	        ELSIF
	            #sx_PreStartManual                                                          // IF in manual jog mode
	            AND (NOT #iq_UDT_EquipmentControl.Request.SignalingRequest                  // Signaling request done
	            OR #Jog_Enable.qx_DelayedSignal)
	            AND NOT #sx_CombinedJogUp                                                   // If selected jog in positive direction
	            AND #sx_CombinedJogDown                                                     // and there is command to jog in negative direction
	        THEN

	            #sx_JogUp := FALSE;                                                         // reset jog positive
	            #sx_JogDown := TRUE;                                                        // set jog negative
	            #sx_Jog := true;

	        ELSIF
	            NOT #sx_PreStartManual                                                      // If not in manual mode
	            OR (#sx_PreStartManual                                                      // or in manual mode
	            AND (#sx_CombinedJogUp                                                      // and jog positive is off
	            AND #sx_CombinedJogDown)                                                    // AND jog negative is off
	            OR (NOT #sx_CombinedJogUp                                                   // or jog positive is on
	            AND NOT #sx_CombinedJogDown))                                               // and jog negative is on
	        THEN

	            #sx_JogUp := FALSE;                                                         // reset jog positive
	            #sx_JogDown := FALSE;                                                       // reset jog negative
	            #sx_Jog := False;
	        END_IF;

	    END_REGION

	END_REGION

	REGION 7 - Semi automatic

	    REGION 7.1 - Semi automatic

	        IF #sx_SemiAutomatic                                                            // Not running Semi-Automatic
	            AND (#ix_ChangeModeSignal
	            AND #ii_Mode = #ci_InfeedMode)
	            AND #sx_SwitchEnable
	            AND NOT #ix_ChuteUpSensor
	        THEN

	            #sx_PreStartSemiAutomaticUp := TRUE;

	            #sx_DownRequest := FALSE;                                                   // Reset down command
	            #sx_UpRequest := TRUE;                                                      // Set up command

	        END_IF;

	        IF #sx_SemiAutomatic                                                            // Not running Semi-Automatic
	            AND (#ix_ChangeModeSignal
	            AND #ii_Mode = #ci_OutfeedMode)
	            AND #sx_SwitchEnable
	            AND NOT #ix_ChuteDownSensor
	        THEN

	            #sx_PreStartSemiAutomaticDown := TRUE;

	            #sx_DownRequest := TRUE;                                                    // Reset down command
	            #sx_UpRequest := FALSE;                                                     // Set up command

	        END_IF;

	        #R_TRIG_PreStartSemiAutomaticUp(CLK := #sx_PreStartSemiAutomaticUp);
	        #R_TRIG_PreStartSemiAutomaticDown(CLK := #sx_PreStartSemiAutomaticDown);

	        //Set Signaling Request
	        IF #R_TRIG_PreStartSemiAutomaticUp.Q OR #R_TRIG_PreStartSemiAutomaticDown.Q THEN
	            #iq_UDT_EquipmentControl.Request.SignalingRequest := TRUE;
	        END_IF;

	        IF #sx_SemiAutomatic
	            AND (#ix_ChuteUpSensor
	            AND #sx_UpRequest)
	            OR #s_UDT_HMIStatus.Specific.SwitchingTimerError
	        THEN
	            #sx_UpRequest := false;
	            #sx_PreStartSemiAutomaticUp := false;
	        END_IF;

	        IF #sx_SemiAutomatic
	            AND (NOT #ix_LiftDownSensor
	            AND #sx_DownRequest)
	            OR #s_UDT_HMIStatus.Specific.SwitchingTimerError
	        THEN
	            #sx_DownRequest := false;
	            #sx_PreStartSemiAutomaticDown := false;
	        END_IF;

	    END_REGION

	    REGION 7.2 - Stop conveyor

	        #qx_ExternalHold := #ss_ColumLiftInterface.Positioning;                                            // External stop signal

	    END_REGION

	END_REGION

	REGION 8 - Write interface DB signals

	    REGION 8.1 - Signal interface

	        #iq_UDT_LiftInterface.InternalErrorReset := #iq_UDT_EquipmentControl.Command.Reset;      // Write Reset signal to the VFD interface
	        #iq_UDT_LiftInterface.ResetStatistics := #iq_UDT_EquipmentControl.Command.ResetData;     // Write Reset data signal to the VFD interface

	    END_REGION

	    REGION 8.1 - Mode selection

	        #ss_ColumLiftInterface.SemiAutomatic :=
	        (#sx_SemiAutomatic                                                               // Automatic started
	        OR #sx_Stopping);                                                                // stopping is activated Go to default position

	        #ss_ColumLiftInterface.Manual :=                                                         // Manual mode is started
	        #sx_CombinedJogUp                                                           // IF selected jog in positive direction
	        OR #sx_CombinedJogDown;

	    END_REGION

	    REGION 8.2 - Run enable

	        #ss_ColumLiftInterface.RunEnabled :=                                                  // Enable the positioning device to run
	        NOT #iq_UDT_LiftInterface.InternalErrorVFD                               // or there are errors in the VFD
	        AND NOT #sx_ConfigurationError                                                   // configuration is wrong
	        AND #ix_HardwareOk                                                        // or an internal error in the RIO panel occured
	        AND (#ss_ColumLiftInterface.SemiAutomatic                                             // VSU is in semi-automatic mode
	        OR (#ss_ColumLiftInterface.Manual                                                     // manual mode is active
	        AND (#sx_CombinedJogUp                                                           // If selected jog in positive direction
	        OR #sx_CombinedJogDown)))                                                        // If selected jog in negative direction
	        AND NOT #ix_RIONotOnline;                                                       // If we don't have signal from sensors

	    END_REGION

	END_REGION

	REGION 9 - Positions reached

	    // triggers of PEC's down/up
	    #F_TRIG_PECUp(CLK := #ix_ChuteUpSensor);
	    #R_TRIG_PECUp(CLK := #ix_ChuteUpSensor);

	    #F_TRIG_PECDown(CLK := #ix_LiftDownSensor);
	    #R_TRIG_PECDown(CLK := #ix_LiftDownSensor);

	    IF #R_TRIG_PECUp.Q THEN
	        #sx_UpperPositionReached := true;
	    ELSIF (#sx_DownRequest OR #sx_JogDown) AND #F_TRIG_PECUp.Q THEN
	        #sx_UpperPositionReached := false;
	    END_IF;

	    IF #R_TRIG_PECDown.Q THEN
	        #sx_LowerPositionReached := true;
	    ELSIF (#sx_UpRequest OR #sx_JogUp) AND #F_TRIG_PECDown.Q THEN
	        #sx_LowerPositionReached := false;
	    END_IF;

	END_REGION

	REGION 10 - Run up/down

	    // Conditions to run column lift upwards
	    #iq_UDT_LiftInterface.RunRvs := ((#sx_UpRequest AND #sx_SemiAutomatic AND NOT #iq_UDT_EquipmentControl.Request.SignalingRequest)
	    OR #sx_JogUp)
	    AND (NOT #sx_UpperPositionReached OR (#sx_MaintenanceControl AND #sx_JogUp))
	    AND #ss_ColumLiftInterface.RunEnabled
	    AND #ix_LiftUpSensor;

	    // Conditions to run column lift down
	    #iq_UDT_LiftInterface.RunFwd := ((#sx_DownRequest AND #sx_SemiAutomatic AND NOT #iq_UDT_EquipmentControl.Request.SignalingRequest)
	    OR #sx_JogDown)
	    AND #ss_ColumLiftInterface.RunEnabled
	    AND #ix_LiftDownSensor;

	END_REGION

	REGION 11 - Column lift speed

	    IF #ss_ColumLiftInterface.Manual THEN
	        #iq_UDT_LiftInterface.SpeedSetpoint := #i_UDT_ColumnLiftConfiguration.ManualModeSpeed;
	    ELSE
	        #iq_UDT_LiftInterface.SpeedSetpoint := #i_UDT_ColumnLiftConfiguration.NominalSpeedSetPoint;
	    END_IF;

	END_REGION

	REGION 12 - Statistics

	    // Down Time
	    IF #sx_SemiAutomatic                                                                 // Automatic active
	        AND NOT #sx_Ready                                                                // Conveyor not ready
	        OR #iq_UDT_EquipmentControl.Command.ResetData                                    // Reset statistics
	    THEN

	        "FC_Statistics"(ix_Reset := #iq_UDT_EquipmentControl.Command.ResetData,              // Or reset statistics from control
	                        ix_Activate := #sx_SemiAutomatic AND NOT #sx_Ready,                  // VSU is stopped
	                        ix_RTrigActivate := #R_TRIG_DownTime.Q,                              // VSU is stopped triger
	                        iqUDT_Statistics := #iq_UDT_Statistics.DownTime);                   // VSU is stopped statistics
	    END_IF;

	    // Up time
	    IF #sx_SemiAutomatic                                // Automatic active
	        AND #sx_Ready                                   // Ready active
	        OR #iq_UDT_EquipmentControl.Command.ResetData   // Reset statistics
	    THEN
	        "FC_Statistics"(ix_Reset := #iq_UDT_EquipmentControl.Command.ResetData,        // OR reset statistics from control
	                        ix_Activate := #sx_SemiAutomatic AND #sx_Ready,                // VSU is running
	                        ix_RTrigActivate := #R_TRIG_UpTime.Q,                          // VSU running trigger
	                        iqUDT_Statistics := #iq_UDT_Statistics.UpTime);               // VSU running statistics

	    END_IF;

	END_REGION

	REGION 13 - Status

	    #s_UDT_Status.Stopped := #sx_Ready AND NOT #sx_SemiAutomatic AND NOT #sx_Stopping;      // stopped
	    #s_UDT_Status.AutoON := #sx_SemiAutomatic OR #sx_Stopping;                              // Auto On
	    #s_UDT_Status.Halted := FALSE;                                                          // Halted
	    #s_UDT_Status.Dieback := FALSE;                                                         // Die back
	    #s_UDT_Status.Running := (#sx_UpRequest OR #sx_DownRequest) AND #sx_SemiAutomatic;      // Running
	    #s_UDT_Status.ManualRun := #ix_SS_Man AND #iq_UDT_LiftInterface.VFDRunning;            // Manual run
	    #s_UDT_Status.Manual := #ix_SS_Man;                                                     // Manual
	    #s_UDT_Status.EnergySave := FALSE;                                                      // Energy save active
	    #s_UDT_Status.SafetyStop := NOT #ix_SafetyOk;                                           // Safety not ok

	    //   Specific status
	    IF #s_UDT_StatusOld <> #s_UDT_Status                                            // update on change
	    THEN

	        // Set status to status number
	        #s_UDT_HMIStatus.Status := 0;                                               // Initialise status number

	        IF #s_UDT_Status.Running                                                    // Running in semi automatic
	        THEN

	            #s_UDT_HMIStatus.Status := "DB_HMIStatusConfiguration".PositionChangeOngoing;

	        END_IF;

	        IF #s_UDT_Status.Stopped                                                    // Stopped
	        THEN

	            #s_UDT_HMIStatus.Status := "DB_HMIStatusConfiguration".Stopped;

	        END_IF;

	        IF #s_UDT_Status.AutoON                                                   // Dieback
	        THEN

	            #s_UDT_HMIStatus.Status := "DB_HMIStatusConfiguration".AutoON;

	        END_IF;

	        IF #s_UDT_Status.ManualRun                                                  // Manual run
	        THEN

	            #s_UDT_HMIStatus.Status := "DB_HMIStatusConfiguration".ManualRun;

	        END_IF;

	        IF #s_UDT_Status.Manual                                                     // Manual
	        THEN

	            #s_UDT_HMIStatus.Status := "DB_HMIStatusConfiguration".Manual;

	        END_IF;

	        IF #iq_UDT_LiftInterface.InternalWarningVFD                                  // The VFD has an internal warning

	        THEN

	            #s_UDT_HMIStatus.Status := "DB_HMIStatusConfiguration".Warning;

	        END_IF;

	        IF #s_UDT_Status.Error                                 // The VFD has an internal warning
	        THEN
	            #s_UDT_HMIStatus.Status := "DB_HMIStatusConfiguration".Error;
	        END_IF;

	        IF #s_UDT_Status.SafetyStop                                                 // Safety stop
	        THEN

	            #s_UDT_HMIStatus.Status := "DB_HMIStatusConfiguration".SafetyStop;

	        END_IF;


	        #s_UDT_StatusOld := #s_UDT_Status;                                          // Copy status TO memory
	        #q_UDT_Status := #s_UDT_Status;                                             // Copy status to output

	    END_IF;

	    //Actual position
	    #s_UDT_HMIStatus.Specific.UpperPosition := #ix_ChuteUpSensor;
	    #s_UDT_HMIStatus.Specific.LowerPosition := NOT #ix_LiftDownSensor;                  //Lower position was changed to use limit switch down because of the project specyfic equipment

	    //Limit switch active
	    IF #sx_LiftUpFiltered AND NOT #ix_RIONotOnline THEN

	        #s_UDT_HMIStatus.Specific.LimitSensorUpperPosition := True;

	    END_IF;

	(*    IF NOT #ix_LiftDownSensor THEN

	        #s_UDT_HMIStatus.Specific.LimitSensorLowerPosition := True;

	    END_IF; *)

	    IF #sx_MaintenanceControl THEN

	        #s_UDT_HMIStatus.Specific.MaintenaceModeActive := True;

	    END_IF;

	    #q_UDT_HMIStatus := #s_UDT_HMIStatus;                                       // Copy status to output

	END_REGION

	REGION 14 - Report to control block

	    #iq_UDT_EquipmentControl.Request.InhibitStop := #iq_UDT_EquipmentControl.Request.InhibitStop OR #ss_ColumLiftInterface.Positioning;

	    "FC_EquipmentReport"(iUDT_Status := #s_UDT_Status,
	                         iqUDT_Control := #iq_UDT_EquipmentControl);

	END_REGION

	REGION 15 - Internal errors and warnings reset

	    #iq_UDT_LiftInterface.InternalErrorPEC := FALSE;
	    #iq_UDT_LiftInterface.InternalWarningTracking := FALSE;
	    #iq_UDT_LiftInterface.InternalErrorTracking := FALSE;
	    #iq_UDT_LiftInterface.InternalWarningVFD := FALSE;
	    #iq_UDT_LiftInterface.InternalErrorVFD := FALSE;
	    #iq_UDT_LiftInterface.Disconnected := FALSE;

	END_REGION

END_FUNCTION_BLOCK

FUNCTION_BLOCK "FB_CodingBeltModes"
{ S7_Optimized_Access := 'TRUE' }
VERSION : 0.1
// ATTRIBUTES
// AUTO_NUMBER = True
// BLOCK_NUMBER = 90
// END_ATTRIBUTES
   VAR_INPUT
      i_UDT_Configuration { ExternalAccessible := 'False'; ExternalVisible := 'False'; ExternalWritable := 'False'} : "UDT_CodingBeltModesConfiguration";   // Function configuration
      ii_Displacement { ExternalAccessible := 'False'; ExternalVisible := 'False'; ExternalWritable := 'False'} : Int;   // Conveyor displacement in one PLC cycle [cm]
      ix_KneeButton { ExternalAccessible := 'False'; ExternalVisible := 'False'; ExternalWritable := 'False'} : Bool;   // Knee button
      ix_LabellingMode { ExternalAccessible := 'False'; ExternalVisible := 'False'; ExternalWritable := 'False'} : Bool;   // Local switch Labeling mode
      ix_ContinueMode { ExternalAccessible := 'False'; ExternalVisible := 'False'; ExternalWritable := 'False'} : Bool;   // Local switch Continue mode
      ix_BufferMode { ExternalAccessible := 'False'; ExternalVisible := 'False'; ExternalWritable := 'False'} : Bool;   // Local switch Buffer mode
      ix_LineModeInfeed { ExternalAccessible := 'False'; ExternalVisible := 'False'; ExternalWritable := 'False'} : Bool;   // Interface with main line - bool or new UDT??? Infeed and Outfeed?
      ix_LineModeOutfeed { ExternalAccessible := 'False'; ExternalVisible := 'False'; ExternalWritable := 'False'} : Bool;   // Interface with main line - bool or new UDT??? Infeed and Outfeed?
      ix_PEC_BoS { ExternalAccessible := 'False'; ExternalVisible := 'False'; ExternalWritable := 'False'} : Bool;   // BoS sensor
      ix_PEC_EoS { ExternalAccessible := 'False'; ExternalVisible := 'False'; ExternalWritable := 'False'} : Bool;   // EoS sensor
   END_VAR

   VAR_OUTPUT
      q_UDT_HMIStatus { ExternalAccessible := 'False'; ExternalVisible := 'False'; ExternalWritable := 'False'} : "UDT_CodingBeltModesStatus";   // Status
      qx_RequestHold_Conveyor { ExternalAccessible := 'False'; ExternalVisible := 'False'; ExternalWritable := 'False'} : Bool;   // Request hold for conveyor
   END_VAR

   VAR
      R_TRIG_KneeButton {InstructionName := 'R_TRIG'; LibVersion := '1.0'; ExternalAccessible := 'False'; ExternalVisible := 'False'; ExternalWritable := 'False'; S7_SetPoint := 'False'} : R_TRIG;   // Rising edge trigger of toogle button
      R_TRIG_LabellingMode {InstructionName := 'R_TRIG'; LibVersion := '1.0'; ExternalAccessible := 'False'; ExternalVisible := 'False'; ExternalWritable := 'False'; S7_SetPoint := 'False'} : R_TRIG;   // Rising edge trigger of labelling mode
      R_TRIG_ContinueMode {InstructionName := 'R_TRIG'; LibVersion := '1.0'; ExternalAccessible := 'False'; ExternalVisible := 'False'; ExternalWritable := 'False'; S7_SetPoint := 'False'} : R_TRIG;   // Rising edge trigger of continue mode
      R_TRIG_BufferMode {InstructionName := 'R_TRIG'; LibVersion := '1.0'; ExternalAccessible := 'False'; ExternalVisible := 'False'; ExternalWritable := 'False'; S7_SetPoint := 'False'} : R_TRIG;   // Rising edge trigger of buffer mode
      R_TRIG_LineModeInfeed {InstructionName := 'R_TRIG'; LibVersion := '1.0'; ExternalAccessible := 'False'; ExternalVisible := 'False'; ExternalWritable := 'False'; S7_SetPoint := 'False'} : R_TRIG;   // Rising edge trigger of Infeed mode
      R_TRIG_LineModeOutfeed {InstructionName := 'R_TRIG'; LibVersion := '1.0'; ExternalAccessible := 'False'; ExternalVisible := 'False'; ExternalWritable := 'False'; S7_SetPoint := 'False'} : R_TRIG;   // Rising edge trigger of Outfeed mode
      F_TRIG_PEC_BoS {InstructionName := 'F_TRIG'; LibVersion := '1.0'; ExternalAccessible := 'False'; ExternalVisible := 'False'; ExternalWritable := 'False'; S7_SetPoint := 'False'} : F_TRIG;   // Falling edge trigger of sensor
      F_TRIG_PEC_EoS {InstructionName := 'F_TRIG'; LibVersion := '1.0'; ExternalAccessible := 'False'; ExternalVisible := 'False'; ExternalWritable := 'False'; S7_SetPoint := 'False'} : F_TRIG;
      sx_LabellingMode { ExternalAccessible := 'False'; ExternalVisible := 'False'; ExternalWritable := 'False'} : Bool;   // Labelling Mode
      sx_ContinueMode { ExternalAccessible := 'False'; ExternalVisible := 'False'; ExternalWritable := 'False'} : Bool;   // Continue Mode
      sx_BufferMode { ExternalAccessible := 'False'; ExternalVisible := 'False'; ExternalWritable := 'False'} : Bool;   // Buffer Mode
      sx_RequestHold { ExternalAccessible := 'False'; ExternalVisible := 'False'; ExternalWritable := 'False'} : Bool;   // Request hold for conveyor
      sx_GeneralError { ExternalAccessible := 'False'; ExternalVisible := 'False'; ExternalWritable := 'False'} : Bool;   // General error
      sx_ConfigurationError { ExternalAccessible := 'False'; ExternalVisible := 'False'; ExternalWritable := 'False'} : Bool;   // Configuration error
      sx_CountDistance { ExternalAccessible := 'False'; ExternalVisible := 'False'; ExternalWritable := 'False'} : Bool;   // Start counting distance to stop position
      sx_ParcelAtPosition { ExternalAccessible := 'False'; ExternalVisible := 'False'; ExternalWritable := 'False'} : Bool;   // The parcel has reached the position
      si_DistanceToStopPosition { ExternalAccessible := 'False'; ExternalVisible := 'False'; ExternalWritable := 'False'} : Int;   // Distance to stop position
   END_VAR


BEGIN
	(*
	----------------------------------------------------------------------------------------
	|                                                                                      |
	|  Copyright  2023             Fortna Europe BV                                        |
	|  All Rights Reserved         Netherlands                                             |
	|                                                                                      |
	|                                                                                      |
	----------------------------------------------------------------------------------------

	Version history:
	Date        | Version   | Author       | Remark
	----------------------------------------------------------------------------------------
	27/07/2023  | 1.0       | S. Nikodem   | Release TIA 17  | DHL Munich 2023
	06/10/2023  | 1.1       | M.Diebel     | Status handling | DHL Munich 2023
	04.12/2023  | 1.2       | M.Diebel     | Stop status     | DHL Munich 2023
	12/03/2024  | 1.3       | S. Nieswiec  | Added to new Baseline
	*)

	REGION 1 - Triggers

	    //Knee button
	    #R_TRIG_KneeButton(CLK := (#ix_KneeButton));

	    //Detect end of the parcel
	    //BoS
	    #F_TRIG_PEC_BoS(CLK := #ix_PEC_BoS);
	    //EoS
	    #F_TRIG_PEC_EoS(CLK := #ix_PEC_EoS);

	END_REGION

	REGION 2 - Error detection

	    // Only one mode can be active
	    IF (#ix_LabellingMode AND #ix_ContinueMode)
	        OR (#ix_LabellingMode AND #ix_BufferMode)
	        OR (#ix_ContinueMode AND #ix_BufferMode)
	    THEN

	        #sx_GeneralError := TRUE;

	    ELSE

	        #sx_GeneralError := False;

	    END_IF;

	    //Configuration Error
	    IF #i_UDT_Configuration.LabellingMode_ParcelStop <= 0 THEN

	        #sx_ConfigurationError := TRUE;

	    ELSE

	        #sx_ConfigurationError := False;

	    END_IF;

	END_REGION

	REGION 3 - Modes

	    // Select mode - when the local switch is used or the main line mode is changed

	    #R_TRIG_LabellingMode(CLK := #ix_LabellingMode AND NOT #sx_BufferMode);

	    #R_TRIG_ContinueMode(CLK := #ix_ContinueMode);

	    #R_TRIG_BufferMode(CLK := #ix_BufferMode AND NOT #sx_LabellingMode);

	    #R_TRIG_LineModeInfeed(CLK := #ix_LineModeInfeed);

	    #R_TRIG_LineModeOutfeed(CLK := #ix_LineModeOutfeed);

	    IF #R_TRIG_LabellingMode.Q
	        OR #R_TRIG_ContinueMode.Q
	        OR #R_TRIG_BufferMode.Q
	        OR #R_TRIG_LineModeInfeed.Q
	        OR #R_TRIG_LineModeOutfeed.Q
	    THEN

	        //Clean value from variable when new mode is selected.
	        #sx_LabellingMode := FALSE;
	        #sx_ContinueMode := FALSE;
	        #sx_BufferMode := FALSE;

	        #sx_CountDistance := FALSE;
	        #si_DistanceToStopPosition := 0;
	        #sx_ParcelAtPosition := FALSE;
	        #sx_RequestHold := FALSE;

	        //
	        IF #ix_LabellingMode AND
	            ((#i_UDT_Configuration.Infeed.LabellingMode AND #ix_LineModeInfeed)
	            OR (#i_UDT_Configuration.Outfeed.LabellingMode AND #ix_LineModeOutfeed))
	        THEN

	            #sx_LabellingMode := True;

	        ELSIF
	            #ix_ContinueMode AND
	            ((#i_UDT_Configuration.Infeed.ContinueMode AND #ix_LineModeInfeed)
	            OR (#i_UDT_Configuration.Outfeed.ContinueMode AND #ix_LineModeOutfeed))
	        THEN

	            #sx_ContinueMode := True;

	        ELSIF
	            #ix_BufferMode AND
	            ((#i_UDT_Configuration.Infeed.BufferMode AND #ix_LineModeInfeed)
	            OR (#i_UDT_Configuration.Outfeed.BufferMode AND #ix_LineModeOutfeed))
	        THEN

	            #sx_BufferMode := True;

	        END_IF;

	    END_IF;

	    REGION 3.1 - Labelling mode

	        IF #sx_LabellingMode THEN

	            IF (#F_TRIG_PEC_BoS.Q AND #ix_LineModeInfeed) OR (#F_TRIG_PEC_EoS.Q AND #ix_LineModeOutfeed) THEN

	                #sx_CountDistance := TRUE;

	            END_IF;

	            //Count the distance to stop parcel position
	            IF #sx_CountDistance THEN

	                #si_DistanceToStopPosition += ABS(#ii_Displacement);

	                IF #si_DistanceToStopPosition > #i_UDT_Configuration.LabellingMode_ParcelStop THEN

	                    #sx_CountDistance := FALSE;
	                    #si_DistanceToStopPosition := 0;
	                    #sx_ParcelAtPosition := True;

	                END_IF;

	            END_IF;

	            //When parcel is at position then stop conveyor
	            #sx_RequestHold := #sx_ParcelAtPosition;

	            //Operator confirm the parcel using knee button
	            IF #R_TRIG_KneeButton.Q THEN

	                #sx_ParcelAtPosition := False;

	            END_IF;


	        END_IF;

	    END_REGION

	    REGION 3.2 - Continue mode

	        IF #sx_ContinueMode THEN

	            IF #R_TRIG_KneeButton.Q THEN

	                #sx_RequestHold := NOT #sx_RequestHold;

	            END_IF;

	        END_IF;

	    END_REGION
	END_REGION

	REGION 4 - Status

	    //Selected mode
	    #q_UDT_HMIStatus.Specific.Infeed_LabellingMode := #sx_LabellingMode AND #ix_LineModeInfeed;
	    #q_UDT_HMIStatus.Specific.Infeed_ContinueMode := #sx_ContinueMode AND #ix_LineModeInfeed;
	    #q_UDT_HMIStatus.Specific.Infeed_BufferMode := #sx_BufferMode AND #ix_LineModeInfeed;
	    #q_UDT_HMIStatus.Specific.Outfeed_LabellingMode := #sx_LabellingMode AND #ix_LineModeOutfeed;
	    #q_UDT_HMIStatus.Specific.Outfeed_ContinueMode := #sx_ContinueMode AND #ix_LineModeOutfeed;
	    #q_UDT_HMIStatus.Specific.Outfeed_BufferMode := #sx_BufferMode AND #ix_LineModeOutfeed;

	    IF (#sx_LabellingMode AND #ix_LineModeInfeed) OR (#sx_LabellingMode AND #ix_LineModeOutfeed)
	    THEN

	        #q_UDT_HMIStatus.Status := "DB_HMIStatusConfiguration".LabbelingMode;

	    END_IF;

	    IF (#sx_ContinueMode AND #ix_LineModeInfeed) OR (#sx_ContinueMode AND #ix_LineModeOutfeed)
	    THEN

	        #q_UDT_HMIStatus.Status := "DB_HMIStatusConfiguration".ContinuousMode;

	    END_IF;

	    IF (#sx_BufferMode AND #ix_LineModeInfeed) OR (#sx_BufferMode AND #ix_LineModeOutfeed)
	    THEN

	        #q_UDT_HMIStatus.Status := "DB_HMIStatusConfiguration".BufferMode;

	    END_IF;

	    IF (NOT #sx_BufferMode AND NOT #sx_ContinueMode AND NOT #sx_LabellingMode AND NOT #ix_LineModeInfeed AND NOT #ix_LineModeOutfeed)
	    THEN

	        #q_UDT_HMIStatus.Status := "DB_HMIStatusConfiguration".Stopped;

	    END_IF;

	    //Errors
	    #q_UDT_HMIStatus.Specific.GeneralError := #sx_GeneralError;
	    #q_UDT_HMIStatus.Specific.ConfigurationError := #sx_ConfigurationError;

	END_REGION

	REGION 5 - Write Output

	    #qx_RequestHold_Conveyor := #sx_RequestHold;

	END_REGION


END_FUNCTION_BLOCK

FUNCTION_BLOCK "FB_Xray_SerialCommunication_Receive"
{ S7_Optimized_Access := 'TRUE' }
VERSION : 0.1
// ATTRIBUTES
// AUTO_NUMBER = True
// BLOCK_NUMBER = 247
// END_ATTRIBUTES
   VAR_INPUT
      i_UDT_SerialCommunicationConfiguration { ExternalAccessible := 'False'; ExternalVisible := 'False'; ExternalWritable := 'False'} : "UDT_SerialComConfiguration";   // Serial communication configuration
      is_ActualTime { ExternalAccessible := 'False'; ExternalVisible := 'False'; ExternalWritable := 'False'} : String;   // Actual date and time in String
      ii_SourceNode { ExternalAccessible := 'False'; ExternalVisible := 'False'; ExternalWritable := 'False'} : Int;   // ID Source Node
      ii_DestinationNode { ExternalAccessible := 'False'; ExternalVisible := 'False'; ExternalWritable := 'False'} : Int;   // ID Destination Node
   END_VAR

   VAR_OUTPUT
      q_UDT_Status { ExternalAccessible := 'False'; ExternalVisible := 'False'; ExternalWritable := 'False'} : "UDT_SerialCommunicationReceiveStatus";   // Status structure
   END_VAR

   VAR_IN_OUT
      iq_UDT_FifoHeader : "UDT_FifoHeader";   // FIFO header
      iqa_FifoData : Array[*] of "UDT_MessageV2";   // FIFO data buffer
      iqi_MessageSequenceNumber { ExternalAccessible := 'False'; ExternalVisible := 'False'; ExternalWritable := 'False'} : Int;   // Message number
   END_VAR

   VAR
      FB_MFC_Sort_COY_ReceiveResult_Instance { ExternalAccessible := 'False'; ExternalVisible := 'False'; ExternalWritable := 'False'; S7_SetPoint := 'False'} : "FB_MFC_Sort_COY_ReceiveResult";   // MFC message generation
      FB_MFC_Sort_COY_Result_Instance { ExternalAccessible := 'False'; ExternalVisible := 'False'; ExternalWritable := 'False'; S7_SetPoint := 'False'} : "FB_MFC_Sort_COY_Result";
      s_Receive_P2P {InstructionName := 'Receive_P2P'; LibVersion := '4.1'; ExternalAccessible := 'False'; ExternalVisible := 'False'; ExternalWritable := 'False'; S7_SetPoint := 'False'} : Receive_P2P;   // PtP receive standard function
      ss_Status { ExternalAccessible := 'False'; ExternalVisible := 'False'; ExternalWritable := 'False'; S7_SetPoint := 'False'} : "UDT_SerialCommunicationReceiveStatus";   // Status structure
      sa_ReceivedMessage { ExternalAccessible := 'False'; ExternalVisible := 'False'; ExternalWritable := 'False'} : Array[1..71] of Char;   // Received a message in Array of chars format
      ss_MessageStructure { ExternalAccessible := 'False'; ExternalVisible := 'False'; ExternalWritable := 'False'} : Struct   // Received a message structure
         EOT { ExternalAccessible := 'False'; ExternalVisible := 'False'; ExternalWritable := 'False'} : String;   // Message structure
         PieceID { ExternalAccessible := 'False'; ExternalVisible := 'False'; ExternalWritable := 'False'} : String;   // Piece ID
         VID { ExternalAccessible := 'False'; ExternalVisible := 'False'; ExternalWritable := 'False'} : String;   // VID
         RoutingCode { ExternalAccessible := 'False'; ExternalVisible := 'False'; ExternalWritable := 'False'} : String;   // RoutingCode
         Group { ExternalAccessible := 'False'; ExternalVisible := 'False'; ExternalWritable := 'False'} : Char;   // Group
         Level { ExternalAccessible := 'False'; ExternalVisible := 'False'; ExternalWritable := 'False'} : Char;   // Level
         Result { ExternalAccessible := 'False'; ExternalVisible := 'False'; ExternalWritable := 'False'} : Char;   // Result
         SOT { ExternalAccessible := 'False'; ExternalVisible := 'False'; ExternalWritable := 'False'} : String;   // SOT
      END_STRUCT;
      ss_Counter { ExternalAccessible := 'False'; ExternalVisible := 'False'; ExternalWritable := 'False'} : Struct   // Counterts only for statistics
         RecivedMessage { ExternalAccessible := 'False'; ExternalVisible := 'False'; ExternalWritable := 'False'} : ULInt;   // Counter of recived message
         CorrectLength { ExternalAccessible := 'False'; ExternalVisible := 'False'; ExternalWritable := 'False'} : ULInt;   // Counter of recived message with correct lenght
         IncorrectLength { ExternalAccessible := 'False'; ExternalVisible := 'False'; ExternalWritable := 'False'} : ULInt;   // Counter of recived message with incorrect lenght
         IncorrectStructure { ExternalAccessible := 'False'; ExternalVisible := 'False'; ExternalWritable := 'False'} : ULInt;   // Counter of recived message with incorrect structure
      END_STRUCT;
      ss_ReceivedMessage { ExternalAccessible := 'False'; ExternalVisible := 'False'; ExternalWritable := 'False'} : String;   // Received a message in String format
      sx_MessageRecived { ExternalAccessible := 'False'; ExternalVisible := 'False'; ExternalWritable := 'False'} : Bool;   // TRUE when new message recived
   END_VAR

   VAR_TEMP
      tui_Cnt : UInt;   // Number of moved characters
      ti_LoopGIN : Int;   // Loop counter - to scan DB_GIN
      ti_LoopTimeout : Int;   // Loop counter - to scan DB_GIN
      tt_TimeDifference : LTime;   // Time difference
      ts_Time1 : String;   // Time value
      ts_Time2 : String;   // Time value
   END_VAR

   VAR CONSTANT
      cs_SOT : String := 'ABC';   // Message constans - SOT
      cc_Underscore : Char := '_';   // Message constans - underscore
      cs_EOT : String := 'XYZ$R$L';   // Message constans - EOT
   END_VAR


BEGIN
	(*
	----------------------------------------------------------------------------------------
	|                                                                                      |
	|  Copyright  2023             FORTNA Europe BV                                        |
	|  All Rights Reserved         Netherlands                                             |
	|                                                                                      |
	----------------------------------------------------------------------------------------
	Version history:
	Date        | Version   | Author       | Remark
	----------------------------------------------------------------------------------------
	27/04/2023  | 1.0       | S. Nikodem   | Release TIA 17 | DHL Munich 2023
	05/10/2023  | 1.1       | S. Nikodem   | Add MFc message generation
	13/03/2024  | 1.2       | S. Nieswiec  | Added to new baseline
	*)

	REGION 1 - Receive

	    #s_Receive_P2P("PORT" := #i_UDT_SerialCommunicationConfiguration."Port",
	                   BUFFER := #ss_ReceivedMessage,
	                   NDR => #ss_Status.NRD,
	                   ERROR => #ss_Status.Erro,
	                   STATUS => #ss_Status.Status,
	                   LENGTH => #ss_Status.Leng);

	    //Check received message lenght
	    IF #ss_Status.NRD THEN

	        //Only for statistics
	        #ss_Counter.RecivedMessage += 1;

	        IF #ss_Status.Leng = #i_UDT_SerialCommunicationConfiguration.ReceiveMessageLength THEN

	            #sx_MessageRecived := True;

	            //Only for statistics
	            #ss_Counter.CorrectLength += 1;

	        ELSE

	            //Only for statistics
	            #ss_Counter.IncorrectLength += 1;

	        END_IF;

	    END_IF;

	END_REGION

	REGION 5- Decode

	    IF #sx_MessageRecived THEN

	        Strg_TO_Chars(Strg := #ss_ReceivedMessage,
	                      pChars := 0,
	                      Cnt => #tui_Cnt,
	                      Chars := #sa_ReceivedMessage);

	        //Combine SOT characters
	        #ss_MessageStructure.SOT := CONCAT(IN1 := #sa_ReceivedMessage[1], IN2 := #sa_ReceivedMessage[2], IN3 := #sa_ReceivedMessage[3]);

	        //Combine EOT characters
	        #ss_MessageStructure.EOT := CONCAT(IN1 := #sa_ReceivedMessage[25],
	                                           IN2 := #sa_ReceivedMessage[26],
	                                           IN3 := #sa_ReceivedMessage[27],
	                                           IN4 := #sa_ReceivedMessage[28],
	                                           IN5 := #sa_ReceivedMessage[29]);


	        IF (#ss_MessageStructure.SOT = #cs_SOT)
	            AND (#ss_MessageStructure.EOT = #cs_EOT)
	        THEN

	            //Piece ID
	            #ss_MessageStructure.PieceID := CONCAT(IN1 := #sa_ReceivedMessage[4],
	                                                   IN2 := #sa_ReceivedMessage[5],
	                                                   IN3 := #sa_ReceivedMessage[6],
	                                                   IN4 := #sa_ReceivedMessage[7],
	                                                   IN5 := #sa_ReceivedMessage[8],
	                                                   IN6 := #sa_ReceivedMessage[9],
	                                                   IN7 := #sa_ReceivedMessage[10],
	                                                   IN8 := #sa_ReceivedMessage[11],
	                                                   IN9 := #sa_ReceivedMessage[12],
	                                                   IN10 := #sa_ReceivedMessage[13],
	                                                   IN11 := #sa_ReceivedMessage[14],
	                                                   IN12 := #sa_ReceivedMessage[15],
	                                                   IN13 := #sa_ReceivedMessage[16],
	                                                   IN14 := #sa_ReceivedMessage[17],
	                                                   IN15 := #sa_ReceivedMessage[18],
	                                                   IN16 := #sa_ReceivedMessage[19],
	                                                   IN17 := #sa_ReceivedMessage[20],
	                                                   IN18 := #sa_ReceivedMessage[21],
	                                                   IN19 := #sa_ReceivedMessage[22],
	                                                   IN20 := #sa_ReceivedMessage[23],
	                                                   IN21 := #sa_ReceivedMessage[24],
	                                                   IN22 := #sa_ReceivedMessage[25],
	                                                   IN23 := #sa_ReceivedMessage[26],
	                                                   IN24 := #sa_ReceivedMessage[27],
	                                                   IN25 := #sa_ReceivedMessage[28],
	                                                   IN26 := #sa_ReceivedMessage[29],
	                                                   IN27 := #sa_ReceivedMessage[30],
	                                                   IN28 := #sa_ReceivedMessage[31],
	                                                   IN29 := #sa_ReceivedMessage[32],
	                                                   IN30 := #sa_ReceivedMessage[33],
	                                                   IN31 := #sa_ReceivedMessage[34],
	                                                   IN32 := #sa_ReceivedMessage[35]);

	            #ss_MessageStructure.PieceID := CONCAT(IN1 := #ss_MessageStructure.PieceID,
	                                                   IN2 := #sa_ReceivedMessage[36],
	                                                   IN3 := #sa_ReceivedMessage[37],
	                                                   IN4 := #sa_ReceivedMessage[38],
	                                                   IN5 := #sa_ReceivedMessage[39],
	                                                   IN6 := #sa_ReceivedMessage[40],
	                                                   IN7 := #sa_ReceivedMessage[41],
	                                                   IN8 := #sa_ReceivedMessage[42],
	                                                   IN9 := #sa_ReceivedMessage[43]);

	            //VID
	            #ss_MessageStructure.VID := CONCAT(IN1 := #sa_ReceivedMessage[45],
	                                               IN2 := #sa_ReceivedMessage[46],
	                                               IN3 := #sa_ReceivedMessage[47],
	                                               IN4 := #sa_ReceivedMessage[48],
	                                               IN5 := #sa_ReceivedMessage[49],
	                                               IN6 := #sa_ReceivedMessage[50],
	                                               IN7 := #sa_ReceivedMessage[51],
	                                               IN8 := #sa_ReceivedMessage[52],
	                                               IN9 := #sa_ReceivedMessage[53],
	                                               IN10 := #sa_ReceivedMessage[54],
	                                               IN11 := #sa_ReceivedMessage[55],
	                                               IN12 := #sa_ReceivedMessage[56],
	                                               IN13 := #sa_ReceivedMessage[57],
	                                               IN14 := #sa_ReceivedMessage[58],
	                                               IN15 := #sa_ReceivedMessage[59],
	                                               IN16 := #sa_ReceivedMessage[60]);

	            //Routing Code
	            #ss_MessageStructure.RoutingCode := CONCAT(IN1 := #sa_ReceivedMessage[61],
	                                                       IN2 := #sa_ReceivedMessage[62]);

	            //Group
	            #ss_MessageStructure.Group := #sa_ReceivedMessage[63];

	            //Level
	            #ss_MessageStructure.Level := #sa_ReceivedMessage[65];

	            //Result
	            #ss_MessageStructure.Result := #sa_ReceivedMessage[66];

	            //Copy data to DB_GIN structure
	            FOR #ti_LoopGIN := #i_UDT_SerialCommunicationConfiguration.GINRangeStart TO #i_UDT_SerialCommunicationConfiguration.GINRangeEnd DO

	                IF ("DB_GIN".GIN[#ti_LoopGIN].DHL.PieceID = #ss_MessageStructure.PieceID)
	                THEN

	                    //Message reviced
	                    "DB_GIN".GIN[#ti_LoopGIN].DHL.Xray.DecisionMessage.Received := TRUE;

	                    //Save message reviced time
	                    "DB_GIN".GIN[#ti_LoopGIN].DHL.Xray.DecisionMessage.ReceivedTime := #is_ActualTime;

	                    //Routing Code
	                    "DB_GIN".GIN[#ti_LoopGIN].DHL.Xray.RoutingCode := #ss_MessageStructure.RoutingCode;

	                    //Group
	                    "DB_GIN".GIN[#ti_LoopGIN].DHL.Xray.Group := #ss_MessageStructure.Group;

	                    //Level
	                    "DB_GIN".GIN[#ti_LoopGIN].DHL.Xray.Level := #ss_MessageStructure.Level;

	                    //Result
	                    "DB_GIN".GIN[#ti_LoopGIN].DHL.Xray.Result := #ss_MessageStructure.Result;

	                    //Message generation
	                    "DB_GIN".GIN[#ti_LoopGIN].DHL.MFCMessage.Sent.XrayResult := TRUE;

	                    //Exit 'for loop'
	                    EXIT;

	                END_IF;

	            END_FOR;

	            //Generate message to MFC
	            //Based on the received message from Xray, generate a message to MFC

	            #FB_MFC_Sort_COY_ReceiveResult_Instance(is_VID := #ss_MessageStructure.VID,
	                                                    is_PieceID := #ss_MessageStructure.PieceID,
	                                                    is_Group := #ss_MessageStructure.Group,
	                                                    is_Level := #ss_MessageStructure.Level,
	                                                    is_Result := #ss_MessageStructure.Result,
	                                                    ii_SourceNode := #ii_SourceNode,
	                                                    ii_DestinationNode := #ii_DestinationNode,
	                                                    iq_UDT_FifoHeader := #iq_UDT_FifoHeader,
	                                                    iqa_FifoData := #iqa_FifoData,
	                                                    iqi_MessageSequenceNumber := #iqi_MessageSequenceNumber);

	        ELSE

	            #ss_Counter.IncorrectStructure += 1;

	        END_IF;

	        //Reset varaible
	        #sx_MessageRecived := false;

	    END_IF;

	END_REGION

	REGION 3 - Receive message timeout

	    FOR #ti_LoopTimeout := #i_UDT_SerialCommunicationConfiguration.GINRangeStart TO #i_UDT_SerialCommunicationConfiguration.GINRangeEnd DO

	        IF "DB_GIN".GIN[#ti_LoopTimeout].DHL.Xray.BagIDMessage.Received
	            AND NOT "DB_GIN".GIN[#ti_LoopTimeout].DHL.Xray.DecisionMessage.Received
	            AND NOT "DB_GIN".GIN[#ti_LoopTimeout].DHL.Xray.DecisionMessage.NotReceivedOnTime
	        THEN

	            //Delete year, month and day from variable
	            #ts_Time1 := DELETE(IN := "DB_GIN".GIN[#ti_LoopTimeout].DHL.Xray.BagIDMessage.TimeReceived, L := 11, P := 1);
	            #ts_Time2 := DELETE(IN := #is_ActualTime, L := 11, P := 1);

	            //Time difference
	            "FC_TimeDiff"(is_EarlierTimeAsString := #ts_Time1,
	                          is_LaterTimeAsString := #ts_Time2,
	                          qt_TimeDifference => #tt_TimeDifference);

	            //Check response time
	            IF #tt_TimeDifference > #i_UDT_SerialCommunicationConfiguration.ResponseTime THEN

	                //Message not received on time
	                "DB_GIN".GIN[#ti_LoopTimeout].DHL.Xray.DecisionMessage.NotReceivedOnTime := True;

	                //FORTNA internal exception results: T = Time-out receiving result
	                "DB_GIN".GIN[#ti_LoopTimeout].DHL.Xray.Result := 'T';

	                //Generate message to MFC
	                #FB_MFC_Sort_COY_Result_Instance(ii_GINRangeStart := #i_UDT_SerialCommunicationConfiguration.GINRangeStart,
	                                                 ii_GINRangeEnd := #i_UDT_SerialCommunicationConfiguration.GINRangeEnd,
	                                                 is_ObjectID := "DB_GIN".GIN[#ti_LoopTimeout].DHL.ObjectID,
	                                                 ii_SourceNode := #ii_SourceNode,
	                                                 ii_DestinationNode := #ii_DestinationNode,
	                                                 iq_UDT_FifoHeader := #iq_UDT_FifoHeader,
	                                                 iqa_FifoData := #iqa_FifoData,
	                                                 iqi_MessageSequenceNumber := #iqi_MessageSequenceNumber);

	                //Message generation
	                "DB_GIN".GIN[#ti_LoopTimeout].DHL.MFCMessage.Sent.XrayResult := TRUE;

	            END_IF;

	        END_IF;

	    END_FOR;

	END_REGION

END_FUNCTION_BLOCK

FUNCTION_BLOCK "FB_ChuteCapacityControl"
{ S7_Optimized_Access := 'TRUE' }
VERSION : 1.1
// ATTRIBUTES
// AUTO_NUMBER = True
// BLOCK_NUMBER = 89
// END_ATTRIBUTES
   VAR_INPUT
      ix_EnableCapacityControl { ExternalAccessible := 'False'; ExternalVisible := 'False'; ExternalWritable := 'False'} : Bool;   // Enable Capacity Control
      ix_ProductSortedToChute { ExternalAccessible := 'False'; ExternalVisible := 'False'; ExternalWritable := 'False'} : Bool;   // Edge on end of  product sorted to chute signal
      idi_DisplacementConveyor { ExternalAccessible := 'False'; ExternalVisible := 'False'; ExternalWritable := 'False'} : DInt;   // Displacment of conveyor [cm]
      idi_GapBack { ExternalAccessible := 'False'; ExternalVisible := 'False'; ExternalWritable := 'False'} : DInt;   // Gap back [mm]
      i_UDT_CapacityControlConfiguration { ExternalAccessible := 'False'; ExternalVisible := 'False'; ExternalWritable := 'False'} : "UDT_CapacityControlConfiguration";   // Capacity control configuration
   END_VAR

   VAR_OUTPUT
      qx_CapacityControlActive { ExternalAccessible := 'False'; ExternalVisible := 'False'; ExternalWritable := 'False'} : Bool;   // Chute capacity control is active
      qx_ProductInChute { ExternalAccessible := 'False'; ExternalVisible := 'False'; ExternalWritable := 'False'} : Bool;   // Product is in chute
   END_VAR

   VAR_IN_OUT
      iqi_ProductLength { ExternalAccessible := 'False'; ExternalVisible := 'False'; ExternalWritable := 'False'} : Int;   // Product Length [mm]
   END_VAR

   VAR
      sdi_ChuteFilling { ExternalAccessible := 'False'; ExternalVisible := 'False'; ExternalWritable := 'False'} : DInt;   // Chute filling
      R_TRIG_EnableCapacityControl {InstructionName := 'R_TRIG'; LibVersion := '1.0'; ExternalAccessible := 'False'; ExternalVisible := 'False'; ExternalWritable := 'False'; S7_SetPoint := 'False'} : R_TRIG;   // R_Trig enable capacity control
   END_VAR

   VAR_TEMP
      tx_CapacityControlActive : Bool;   // TRUE if Chute filling is more than halfull but isn't full
   END_VAR


BEGIN
	(*
	----------------------------------------------------------------------------------------
	|                                                                                      |
	|  Copyright  2023             FORTNA Europe BV                                        |
	|  All Rights Reserved         Netherlands                                             |
	|                                                                                      |
	----------------------------------------------------------------------------------------

	Version history:
	Date        | Version   | Author            | Remark
	----------------------------------------------------------------------------------------
	 01/03/2023 | 1.0       | R. Golonka       | first release TIA 17.0 | DHL Munich
	 01/03/2023 | 1.1       | S.Theocharis     | Add absolute instruction for displacement
	 12/03/2024 | 1.2       | S. Nieswiec      | Added to new Baseline
	 *)

	REGION 1 - Inicialization
	    // Reset outputs and status
	    IF NOT #ix_EnableCapacityControl THEN
	        #sdi_ChuteFilling := 0;
	        #qx_CapacityControlActive := 0;
	        #qx_ProductInChute := 0;
	        RETURN;
	    END_IF;

	    // Rising trig after enable
	    #R_TRIG_EnableCapacityControl(CLK := #ix_EnableCapacityControl);

	    // Set zero to chute filing at first scan or function enable
	    IF "DB_Memory".FirstScan OR #R_TRIG_EnableCapacityControl.Q
	    THEN
	        #sdi_ChuteFilling := 0;
	    END_IF;

	END_REGION

	REGION 2 - Chute filling count down
	    // Count chute filling with conveyor displacement
	    IF (#idi_DisplacementConveyor <> 0) AND (#sdi_ChuteFilling >= 0)
	    THEN
	        // Chute filing subtract displacement of conveyor [cm to mm]
	        #sdi_ChuteFilling -= (ABS(#idi_DisplacementConveyor) * 10);
	        // Set zero to chute filling
	        IF (#sdi_ChuteFilling < 0)
	        THEN
	            #sdi_ChuteFilling := 0;
	        END_IF;
	    END_IF;
	END_REGION

	REGION 3 - Chute filling count up
	    // Calculate chute filling when product appear (ProductSortedToChute appear for one cycle)
	    IF #ix_ProductSortedToChute AND (#sdi_ChuteFilling >= 0) AND (#sdi_ChuteFilling < #i_UDT_CapacityControlConfiguration.ChuteLength)
	    THEN
	        #sdi_ChuteFilling := #sdi_ChuteFilling + #idi_GapBack + INT_TO_DINT(#iqi_ProductLength);
	        #iqi_ProductLength := 0;
	    END_IF;

	    //Set maximum chute lenght when chute filing is biger than maximum chute lenght
	    IF #sdi_ChuteFilling >= #i_UDT_CapacityControlConfiguration.ChuteLength THEN
	        #sdi_ChuteFilling := #i_UDT_CapacityControlConfiguration.ChuteLength;
	    END_IF;

	END_REGION

	REGION 4 - Capacity control active
	    // Capacity Control is active if chute filling isn't halffull or isn't full
	    #tx_CapacityControlActive :=
	    (#sdi_ChuteFilling > #i_UDT_CapacityControlConfiguration.MaxProductLenght) OR (#sdi_ChuteFilling > #i_UDT_CapacityControlConfiguration.ProductLenghtHalfFull);

	END_REGION

	REGION 5 - Outputs
	    // Set output of capacity control (True when chute don't want more parcel)
	    #qx_CapacityControlActive := #tx_CapacityControlActive;

	    // Product is in Chute
	    #qx_ProductInChute := (#sdi_ChuteFilling > 0);

	END_REGION

	REGION 6 - Status
	    // Status of chute capacity control

	END_REGION


END_FUNCTION_BLOCK

FUNCTION_BLOCK "FB_BiDirectionalControl"
{ S7_Optimized_Access := 'TRUE' }
VERSION : 0.1
// ATTRIBUTES
// AUTO_NUMBER = True
// BLOCK_NUMBER = 88
// END_ATTRIBUTES
   VAR_INPUT
      i_UDT_BiDirectionalConfguration { ExternalAccessible := 'False'; ExternalVisible := 'False'; ExternalWritable := 'False'} : "UDT_BiDirectionalConfiguration";   // Configuration structure
      ii_SystemMode { ExternalAccessible := 'False'; ExternalVisible := 'False'; ExternalWritable := 'False'} : Int;   // System mode message from MFC
      ix_EmptyInfeedLine { ExternalAccessible := 'False'; ExternalVisible := 'False'; ExternalWritable := 'False'} : Bool;   // Empty infeed line
      ix_EmptyOutfeedLine { ExternalAccessible := 'False'; ExternalVisible := 'False'; ExternalWritable := 'False'} : Bool;   // Empty outfeed line
   END_VAR

   VAR_OUTPUT
      q_UDT_HMIStatus { ExternalAccessible := 'False'; ExternalVisible := 'False'; ExternalWritable := 'False'} : "UDT_BiDirectionalStatus";   // Status structure
   END_VAR

   VAR_IN_OUT
      iq_UDT_InfeedSystem : "UDT_EquipmentControl";   // Infeed system equipment control
      iq_UDT_OutfeedSystem : "UDT_EquipmentControl";   // Outfeed system equipment control
      iq_UDT_BiDirectionalInterface : "UDT_BiDirectionalInterface";   // BiDirectional function inteface structure
   END_VAR

   VAR
      R_TRIG_InfeedMode {InstructionName := 'R_TRIG'; LibVersion := '1.0'; ExternalAccessible := 'False'; ExternalVisible := 'False'; ExternalWritable := 'False'; S7_SetPoint := 'False'} : R_TRIG;   // Rising edge trigger of infeed mode
      R_TRIG_OutfeedMode {InstructionName := 'R_TRIG'; LibVersion := '1.0'; ExternalAccessible := 'False'; ExternalVisible := 'False'; ExternalWritable := 'False'; S7_SetPoint := 'False'} : R_TRIG;   // Rising edge trigger of outfeed mode
      R_TRIG_OutfeedStopped {InstructionName := 'R_TRIG'; LibVersion := '1.0'; ExternalAccessible := 'False'; ExternalVisible := 'False'; ExternalWritable := 'False'; S7_SetPoint := 'False'} : R_TRIG;   // Rising edge trigger of outfeed system stopped
      R_TRIG_InfeedStopped {InstructionName := 'R_TRIG'; LibVersion := '1.0'; ExternalAccessible := 'False'; ExternalVisible := 'False'; ExternalWritable := 'False'; S7_SetPoint := 'False'} : R_TRIG;   // Rising edge trigger of infeed system stopped
   END_VAR
   VAR RETAIN
      s_UDT_HMIStatus { ExternalAccessible := 'False'; ExternalVisible := 'False'; ExternalWritable := 'False'; S7_SetPoint := 'False'} : "UDT_BiDirectionalStatus";   // Status structure
      si_StepNumber { ExternalAccessible := 'False'; ExternalVisible := 'False'; ExternalWritable := 'False'} : Int;   // Step number
   END_VAR

   VAR CONSTANT
      ci_InfeedMode : Int := 1;   // Infeed mode number
      ci_OutfeedMode : Int := 2;   // Outfeed mode number
   END_VAR


BEGIN
	(*
	----------------------------------------------------------------------------------------
	|                                                                                      |
	|  Copyright  2023             FORTNA Europe BV                                        |
	|  All Rights Reserved         Netherlands                                             |
	|                                                                                      |
	----------------------------------------------------------------------------------------

	Version history:
	Date        | Version   | Author       | Remark
	----------------------------------------------------------------------------------------
	20/07/2023  | 1.0       | S. Nikodem   | Release TIA 17 | DHL Munich 2023
	13/12/2023  | 1.1       | S. Nikodem   | Added input time freeze
	13/12/2023  | 1.2       | S. Nikodem   | Update
	17/01/2024  | 1.3       | L. Klar      | Update
	07/02/2024  | 1.3       | L. Klar      | Stop switching device added
	*)

	REGION 1 - Triggers

	    //Infeed mode active
	    #R_TRIG_InfeedMode(CLK := (#ii_SystemMode = #ci_InfeedMode));

	    //Outfeed mode active
	    #R_TRIG_OutfeedMode(CLK := (#ii_SystemMode = #ci_OutfeedMode));

	    //Outfeed system stopped
	    #R_TRIG_OutfeedStopped(CLK := #iq_UDT_BiDirectionalInterface.OutfeedStopped);

	    //Infeed system stopped
	    #R_TRIG_InfeedStopped(CLK := #iq_UDT_BiDirectionalInterface.InfeedStopped);

	END_REGION

	REGION 2 - Select mode

	    //Initial value when mode changed
	    IF (#R_TRIG_OutfeedMode.Q OR #R_TRIG_InfeedMode.Q) AND NOT "DB_Memory".FirstScan THEN

	        //Reset
	        #si_StepNumber := 1;

	        #s_UDT_HMIStatus.InfeedModeRequested := False;
	        #s_UDT_HMIStatus.OutfeedModeRequested := False;
	        #s_UDT_HMIStatus.InfeedModeReady := False;
	        #s_UDT_HMIStatus.OutfeedModeReady := False;
	        #s_UDT_HMIStatus.ChangingMode := False;

	    END_IF;

	    //Proces selected mode
	    CASE #ii_SystemMode OF
	        #ci_InfeedMode://InfeedMode

	            CASE #si_StepNumber OF
	                1: //Requested to change the mode of operation of the system

	                    //Set
	                    #s_UDT_HMIStatus.InfeedModeRequested := TRUE;
	                    #s_UDT_HMIStatus.ChangingMode := TRUE;
	                    #si_StepNumber := 2;

	                2://Waiting for the line to empty, according to the configured time

	                    IF #ix_EmptyOutfeedLine//#s_FB_TimeDelayInfeed.qx_DelayedSignal
	                    THEN
	                        //Set
	                        #iq_UDT_BiDirectionalInterface.RequestToStopOutfeed := TRUE;
	                        #iq_UDT_BiDirectionalInterface.RequestToStopBidirectional := TRUE;
	                        #si_StepNumber := 3;
	                    END_IF;

	                3://Checking if the line stopped

	                    IF #iq_UDT_BiDirectionalInterface.OutfeedStopped THEN
	                        //Reset
	                        #iq_UDT_BiDirectionalInterface.RequestToStopOutfeed := False;
	                        #s_UDT_HMIStatus.OutfeedModeActive := False;
	                    END_IF;
	                    IF #iq_UDT_BiDirectionalInterface.BidirectionalStopped THEN
	                        //Reset
	                        #iq_UDT_BiDirectionalInterface.RequestToStopBidirectional := False;
	                    END_IF;

	                    //Stopping or changing the position of the switching device
	                    IF NOT #iq_UDT_BiDirectionalInterface.RequestToStopOutfeed
	                        AND NOT #iq_UDT_BiDirectionalInterface.RequestToStopBidirectional
	                    THEN
	                        //Set
	                        #iq_UDT_BiDirectionalInterface.RequestToSwitchingSystem := True;
	                        #si_StepNumber := 4;
	                    END_IF;

	                4://Check if Switching system is in position

	                    IF #iq_UDT_BiDirectionalInterface.SwitchingSystemReady
	                    THEN
	                        //Reset
	                        #iq_UDT_BiDirectionalInterface.RequestToSwitchingSystem := FALSE;
	                        #iq_UDT_BiDirectionalInterface.RequestToStopSwitchingSystem := TRUE;
	                        #s_UDT_HMIStatus.InfeedModeRequested := FALSE;
	                        #s_UDT_HMIStatus.ChangingMode := FALSE;

	                        //Set
	                        #s_UDT_HMIStatus.InfeedModeReady := True;
	                        #si_StepNumber := 5;
	                    END_IF;

	                5://The system is ready to restart, waiting for the command.

	                    IF #s_UDT_HMIStatus.InfeedModeReady

	                        AND (#iq_UDT_InfeedSystem.Command.Start
	                        OR #iq_UDT_InfeedSystem.Command.AutomaticOn)
	                    THEN
	                        //Reset
	                        #iq_UDT_BiDirectionalInterface.RequestToStopSwitchingSystem := FALSE;
	                        #s_UDT_HMIStatus.InfeedModeReady := False;
	                        //Set
	                        #s_UDT_HMIStatus.InfeedModeActive := True;
	                    END_IF;

	                    IF (#iq_UDT_InfeedSystem.Command.Stop
	                        OR NOT #iq_UDT_InfeedSystem.Command.AutomaticOn)
	                    THEN
	                        // Set
	                        #s_UDT_HMIStatus.InfeedModeReady := True;

	                    END_IF;

	            END_CASE;

	        #ci_OutfeedMode://OutfeedMode

	            CASE #si_StepNumber OF
	                1://Requested to change the mode of operation of the system

	                    //Set
	                    #s_UDT_HMIStatus.OutfeedModeRequested := TRUE;
	                    #s_UDT_HMIStatus.ChangingMode := TRUE;
	                    #si_StepNumber := 2;


	                2:   //Waiting for the line to empty, according to the configured time

	                    IF #ix_EmptyInfeedLine// #s_FB_TimeDelayOutfeed.qx_DelayedSignal

	                    THEN
	                        #iq_UDT_BiDirectionalInterface.RequestToStopInfeed := TRUE;
	                        #iq_UDT_BiDirectionalInterface.RequestToStopBidirectional := TRUE;
	                        #si_StepNumber := 3;
	                    END_IF;


	                3: //Checking if the line stopped

	                    IF #iq_UDT_BiDirectionalInterface.InfeedStopped THEN
	                        //Reset
	                        #iq_UDT_BiDirectionalInterface.RequestToStopInfeed := False;
	                        #s_UDT_HMIStatus.InfeedModeActive := False;
	                    END_IF;
	                    IF #iq_UDT_BiDirectionalInterface.BidirectionalStopped THEN
	                        //Reset
	                        #iq_UDT_BiDirectionalInterface.RequestToStopBidirectional := False;
	                    END_IF;

	                    //Stopping or changing the position of the switching device
	                    IF NOT #iq_UDT_BiDirectionalInterface.RequestToStopInfeed
	                        AND NOT #iq_UDT_BiDirectionalInterface.RequestToStopBidirectional
	                    THEN
	                        //Set
	                        #iq_UDT_BiDirectionalInterface.RequestToSwitchingSystem := True;
	                        #si_StepNumber := 4;
	                    END_IF;

	                4://Check if Switching system is in position

	                    IF #iq_UDT_BiDirectionalInterface.SwitchingSystemReady
	                    THEN
	                        //Reset
	                        #iq_UDT_BiDirectionalInterface.RequestToSwitchingSystem := FALSE;
	                        #iq_UDT_BiDirectionalInterface.RequestToStopSwitchingSystem := TRUE;
	                        #s_UDT_HMIStatus.OutfeedModeRequested := FALSE;
	                        #s_UDT_HMIStatus.ChangingMode := FALSE;
	                        //Set
	                        #s_UDT_HMIStatus.OutfeedModeReady := True;
	                        #si_StepNumber := 5;
	                    END_IF;

	                5://The system is ready to restart, waiting for the command.

	                    IF #s_UDT_HMIStatus.OutfeedModeReady
	                        AND (#iq_UDT_OutfeedSystem.Command.Start
	                        OR #iq_UDT_OutfeedSystem.Command.AutomaticOn)
	                    THEN
	                        //Reset
	                        #s_UDT_HMIStatus.OutfeedModeReady := False;
	                        #iq_UDT_BiDirectionalInterface.RequestToStopSwitchingSystem := FALSE;
	                        //Set
	                        #s_UDT_HMIStatus.OutfeedModeActive := True;
	                    END_IF;

	                    IF (#iq_UDT_OutfeedSystem.Command.Stop
	                        OR NOT #iq_UDT_OutfeedSystem.Command.AutomaticOn)
	                    THEN
	                        // Set
	                        #s_UDT_HMIStatus.OutfeedModeReady := True;

	                    END_IF;

	            END_CASE;

	    END_CASE;

	END_REGION

	REGION 3 - Status

	    // //Copy time
	    // CASE #ii_SystemMode OF
	    //     1:
	    //         //Convert time from ms to sec
	    //         #iq_UDT_BiDirectionalInterface.ElapsedTime := LREAL_TO_UDINT(#s_FB_TimeDelayInfeed.qlr_ActualTime) / 1000;

	    //         IF #i_UDT_BiDirectionalConfguration.TimeDelayInfeed <= #s_FB_TimeDelayInfeed.qlr_ActualTime THEN
	    //             #iq_UDT_BiDirectionalInterface.ElapsedTime := 0;
	    //         END_IF;

	    //     2:
	    //         //Convert time from ms to sec
	    //         #iq_UDT_BiDirectionalInterface.ElapsedTime := LREAL_TO_UDINT(#s_FB_TimeDelayOutfeed.qlr_ActualTime) / 1000;

	    //         IF #i_UDT_BiDirectionalConfguration.TimeDelayOutfeed <= #s_FB_TimeDelayOutfeed.qlr_ActualTime THEN
	    //             #iq_UDT_BiDirectionalInterface.ElapsedTime := 0;
	    //         END_IF;

	    //     ELSE

	    //         #iq_UDT_BiDirectionalInterface.ElapsedTime := 0;

	    // END_CASE;

	    // //Reset ststem mode status
	    // IF #R_TRIG_OutfeedStopped.Q THEN

	    //     #s_UDT_HMIStatus.OutfeedModeActive := False;

	    // END_IF;

	    // //Reset ststem mode status
	    // IF #R_TRIG_InfeedStopped.Q THEN

	    //     #s_UDT_HMIStatus.InfeedModeActive := False;

	    // END_IF;

	    //Copy starus to output structure
	    #q_UDT_HMIStatus := #s_UDT_HMIStatus;

	END_REGION

END_FUNCTION_BLOCK

FUNCTION_BLOCK "FB_XbeltCommon_Interface"
{ S7_Optimized_Access := 'TRUE' }
VERSION : 1.0
// ATTRIBUTES
// AUTO_NUMBER = True
// BLOCK_NUMBER = 246
// END_ATTRIBUTES
   VAR_INPUT
      i_UDT_Sorter_DownStream_Common { ExternalAccessible := 'False'; ExternalVisible := 'False'; ExternalWritable := 'False'} : "UDT_Sorter_DownStream_Common";   // Sorter Downstream structure
      ix_FireAlarm { ExternalAccessible := 'False'; ExternalVisible := 'False'; ExternalWritable := 'False'} : Bool;   // Fire alarm
   END_VAR

   VAR_OUTPUT
      q_UDT_DownStream_Sorter_Common { ExternalAccessible := 'False'; ExternalVisible := 'False'; ExternalWritable := 'False'} : "UDT_DownStream_Sorter_Common";   // Downstream Sorter structure
      qx_WatchDogError { ExternalAccessible := 'False'; ExternalVisible := 'False'; ExternalWritable := 'False'} : Bool;   // WatchDog error
      qx_AvailableCarriers { ExternalAccessible := 'False'; ExternalVisible := 'False'; ExternalWritable := 'False'} : Bool;   // Available carriers
   END_VAR

   VAR_IN_OUT
      iq_UDT_ConnectStatus : "UDT_ConnectStatus";   // Connect status structure
   END_VAR

   VAR
      s_FB_ConnectionCheck { ExternalAccessible := 'False'; ExternalVisible := 'False'; ExternalWritable := 'False'; S7_SetPoint := 'False'} : "FB_ConnectionCheck";   // FB to connection check
      s_UDT_DownStream_Sorter_Common { ExternalAccessible := 'False'; ExternalVisible := 'False'; ExternalWritable := 'False'; S7_SetPoint := 'False'} : "UDT_DownStream_Sorter_Common";   // static DownStream Sorter
      sx_WatchDogError { ExternalAccessible := 'False'; ExternalVisible := 'False'; ExternalWritable := 'False'} : Bool;   // static WatchDog Error
      sx_AvailableCarriers { ExternalAccessible := 'False'; ExternalVisible := 'False'; ExternalWritable := 'False'} : Bool;   // static available Carriers
   END_VAR


BEGIN

	(*
	----------------------------------------------------------------------------------------
	|                                                                                      |
	|  Copyright  2023             FORTNA Europe BV                                        |
	|  All Rights Reserved         Netherlands                                             |
	|                                                                                      |
	----------------------------------------------------------------------------------------

	Version history:
	Date        | Version   | Author            | Remark
	----------------------------------------------------------------------------------------
	 30/03/2023 | 0.1       | R.Golonka         | first release TIA 17.0 | DHL Munich
	 11/09/2023 | 1.0       | S.Theocharis      | Added watchdog output
	 13/03/2024 | 1.1       | S. Nieswiec       | Added to new baseline
	 *)

	REGION 1 - Fire alarm

	    // Fire alarm
	    #s_UDT_DownStream_Sorter_Common.FireAlarm := #ix_FireAlarm;

	END_REGION

	REGION 2 - Available carriees

	    // Available carriees
	    #sx_AvailableCarriers := (#i_UDT_Sorter_DownStream_Common.AvailableCarriers = 1);

	END_REGION

	REGION 3 - Connection check

	    // Connection status check
	    #s_FB_ConnectionCheck(ib_Watchdog := #i_UDT_Sorter_DownStream_Common.Watchdog,
	                          ix_Trigger100ms := "DB_Memory"."OS_0.1sec",
	                          qb_Watchdog => #s_UDT_DownStream_Sorter_Common.Watchdog,
	                          iqudt_ConnectionStatus := #iq_UDT_ConnectStatus);

	END_REGION

	REGION 4 - Output update

	    // Output update
	    #q_UDT_DownStream_Sorter_Common := #s_UDT_DownStream_Sorter_Common;
	    #qx_AvailableCarriers := #sx_AvailableCarriers;
	    #qx_WatchDogError := #sx_WatchDogError;

	END_REGION


END_FUNCTION_BLOCK

FUNCTION_BLOCK "FB_SNCY_Result"
{ S7_Optimized_Access := 'TRUE' }
VERSION : 0.1
// ATTRIBUTES
// AUTO_NUMBER = True
// BLOCK_NUMBER = 244
// END_ATTRIBUTES
   VAR_INPUT
      ii_DecisionPoint { ExternalAccessible := 'False'; ExternalVisible := 'False'; ExternalWritable := 'False'} : Int;   // Decision Point - Distance from the end of the conveyor
      ii_DischargeLocation { ExternalAccessible := 'False'; ExternalVisible := 'False'; ExternalWritable := 'False'} : UInt;   // Discharge location identifier
      ix_PEC { ExternalAccessible := 'False'; ExternalVisible := 'False'; ExternalWritable := 'False'} : Bool;   // TRUE when PEC is not blocked
   END_VAR

   VAR_IN_OUT
      iqa_TrackingData : Array[*] of Int;   // Conveyor tracking data
      iq_UDT_FifoHeader_MFCMessage : "UDT_FifoHeader";   // MFC Message FIFO header
      iqs_FifoData_MFCMessage : Array[*] of "UDT_MessageV2";   // MFC Message FIFO data buffer
      iqdi_MessageSequenceNumber { ExternalAccessible := 'False'; ExternalVisible := 'False'; ExternalWritable := 'False'} : Int;   // MFC Message Message number
   END_VAR

   VAR
      s_FB_MFC_Sort_SortResult { ExternalAccessible := 'False'; ExternalVisible := 'False'; ExternalWritable := 'False'; S7_SetPoint := 'False'} : "FB_MFC_Sort_SortResult";
   END_VAR


BEGIN
	(*
	----------------------------------------------------------------------------------------
	|                                                                                      |
	|  Copyright  2023             FORTNA Europe BV                                        |
	|  All Rights Reserved         Netherlands                                             |
	|                                                                                      |
	----------------------------------------------------------------------------------------
	Version history:
	Date        | Version   | Author       | Remark
	----------------------------------------------------------------------------------------
	05/07/2023  | 1.0       | S. Nikodem   | Release TIA 17 | DHL Munich 2023
	13/03/2024  | 1.1       | S. Nieswiec  | Added to new baseline, block needs uptade after munich is finished
	02/05/2024  | 1.2       | J.Majer      | Datatype conversions changed from automatic to explicit, to accomodate IEC 61131-3 standard

	*)

	REGION 1 - Combine data

	    IF NOT #ix_PEC
	        AND #iqa_TrackingData[#ii_DecisionPoint] <> 0
	        AND NOT "DB_GIN".GIN[#iqa_TrackingData[#ii_DecisionPoint]].DHL.MFCMessage.Sent.SortResult
	    THEN

	        //Parcel sorted correctly
	        "DB_GIN".GIN[#iqa_TrackingData[#ii_DecisionPoint]].General.SortStatus.GoodDivert := True;
	        "DB_GIN".GIN[#iqa_TrackingData[#ii_DecisionPoint]].General.SortStatus.DivertDestination := UINT_TO_INT(#ii_DischargeLocation);

	        //Sort Result message - parcel sorted correctly
	        #s_FB_MFC_Sort_SortResult(is_ObjectID := "DB_GIN".GIN[#iqa_TrackingData[#ii_DecisionPoint]].DHL.ObjectID,
	                                  ii_DischargeLocation := #ii_DischargeLocation,
	                                  ii_Result := 1,
	                                  ii_Reason := 1,
	                                  iq_UDT_FifoHeader := #iq_UDT_FifoHeader_MFCMessage,
	                                  iqs_FifoData := #iqs_FifoData_MFCMessage,
	                                  iqdi_MessageSequenceNumber := #iqdi_MessageSequenceNumber);

	        //Sort Result message generated
	        "DB_GIN".GIN[#iqa_TrackingData[#ii_DecisionPoint]].DHL.MFCMessage.Sent.SortResult := True;

	    END_IF;

	END_REGION





END_FUNCTION_BLOCK

FUNCTION_BLOCK "FB_LocalMotorControl"
{ S7_Optimized_Access := 'TRUE' }
VERSION : 0.1
// ATTRIBUTES
// AUTO_NUMBER = True
// BLOCK_NUMBER = 98
// END_ATTRIBUTES
   VAR_INPUT
      ix_StartStopButton { ExternalAccessible := 'False'; ExternalVisible := 'False'; ExternalWritable := 'False'} : Bool;   // Local motor control pushbutton
   END_VAR

   VAR_OUTPUT
      qx_PilotLamp { ExternalAccessible := 'False'; ExternalVisible := 'False'; ExternalWritable := 'False'} : Bool;   // Pilot lamp of blue colour
   END_VAR

   VAR_IN_OUT
      iq_UDT_EquipmentControl : "UDT_EquipmentControl";   //           Equipment control structure
      iq_UDT_ConveyorCommand : "UDT_ConveyorCommand";   // Conveyor command stucture
      iq_UDT_ConveyorInterface : "UDT_ConveyorInterface";   // Interface structure
   END_VAR

   VAR
      R_TRIG_ToogleButton {InstructionName := 'R_TRIG'; LibVersion := '1.0'; ExternalAccessible := 'False'; ExternalVisible := 'False'; ExternalWritable := 'False'; S7_SetPoint := 'False'} : R_TRIG;   // Rising edge trigger manual mode
   END_VAR


BEGIN
	(*
	----------------------------------------------------------------------------------------
	|                                                                                      |
	|  Copyright  2023             Fortna Europe BV                                        |
	|  All Rights Reserved         Netherlands                                             |
	|                                                                                      |
	|                                                                                      |
	----------------------------------------------------------------------------------------

	Version history:
	Date        | Version   | Author       | Remark
	----------------------------------------------------------------------------------------
	18/11/2022  | 1.0       | S. Nikodem   | Release TIA 17 | DHL Munich 2023
	07/12/2023  | 1.1       | S. Nikodem   | Added Equipment Control structure
	13/03/2024  | 1.2       | S. Nieswiec  | Added to new Baseline
	*)

	REGION 1  - Pilot blue lamp

	    //Is flash when manual mode is acive and motor is ready to start. When the motor is running then lamp will stay solid
	    #qx_PilotLamp := ((#iq_UDT_ConveyorCommand.ManualMode OR #iq_UDT_EquipmentControl.Command.ManualMode) AND "mx_Clock_1Hz") OR #iq_UDT_ConveyorInterface.VFDRunning;

	END_REGION

	REGION 2 - Toggle button function

	    //One button can start and stop the conveyor
	    //Memory to save information about positive edge
	    #R_TRIG_ToogleButton(CLK := (#ix_StartStopButton));

	    IF #iq_UDT_ConveyorCommand.ManualMode OR #iq_UDT_EquipmentControl.Command.ManualMode THEN
	        IF #R_TRIG_ToogleButton.Q THEN

	            #iq_UDT_ConveyorCommand.ManualStartStop := NOT #iq_UDT_ConveyorCommand.ManualStartStop;

	        END_IF;
	    ELSE
	        //Reset value
	        #iq_UDT_ConveyorCommand.ManualStartStop := 0;

	    END_IF;

	END_REGION
END_FUNCTION_BLOCK

FUNCTION_BLOCK "FB_SNCY_Lost"
{ S7_Optimized_Access := 'TRUE' }
VERSION : 0.1
// ATTRIBUTES
// AUTO_NUMBER = True
// BLOCK_NUMBER = 243
// END_ATTRIBUTES
   VAR_INPUT
      ii_SourceNode { ExternalAccessible := 'False'; ExternalVisible := 'False'; ExternalWritable := 'False'} : Int := 0;   // Source Node
      ii_DestinationNode { ExternalAccessible := 'False'; ExternalVisible := 'False'; ExternalWritable := 'False'} : Int := 0;   // Destination Node
   END_VAR

   VAR_IN_OUT
      iqs_FifoData_LostGin : Array[*] of Int;   //  Lost Gin Fifo data
      iq_UDT_FifoHeader_LostGin : "UDT_FifoHeader";   //  Lost Gin Fifo header
      iq_UDT_FifoHeader_MFCMessage : "UDT_FifoHeader";   // MFC Message FIFO header
      iqs_FifoData_MFCMessage : Array[*] of "UDT_MessageV2";   // MFC Message FIFO data buffer
      iqdi_MessageSequenceNumber { ExternalAccessible := 'False'; ExternalVisible := 'False'; ExternalWritable := 'False'} : Int;   // MFC Message Message number
   END_VAR

   VAR
      s_FB_MFC_Sort_SortResult { ExternalAccessible := 'False'; ExternalVisible := 'False'; ExternalWritable := 'False'; S7_SetPoint := 'False'} : "FB_MFC_Sort_SortResult";   // Message generator
      ss_Status { ExternalAccessible := 'False'; ExternalVisible := 'False'; ExternalWritable := 'False'} : Struct   // FiFo status
         FIFOStatus { ExternalAccessible := 'False'; ExternalVisible := 'False'; ExternalWritable := 'False'; S7_SetPoint := 'False'} : "UDT_FifoStatus";   // Fifo status
         FIFOError { ExternalAccessible := 'False'; ExternalVisible := 'False'; ExternalWritable := 'False'} : Bool;   // Fifo error
         FIFOWarning { ExternalAccessible := 'False'; ExternalVisible := 'False'; ExternalWritable := 'False'} : Bool;   // Fifio warning
         InvalidGIN { ExternalAccessible := 'False'; ExternalVisible := 'False'; ExternalWritable := 'False'} : Bool;   // Invalid GIN
         InvalidMessageLength { ExternalAccessible := 'False'; ExternalVisible := 'False'; ExternalWritable := 'False'} : Bool;   // Invalid message lenght
         InvalidMessagegArraySize { ExternalAccessible := 'False'; ExternalVisible := 'False'; ExternalWritable := 'False'} : Bool;   // Invalid message array size
      END_STRUCT;
      si_GIN { ExternalAccessible := 'False'; ExternalVisible := 'False'; ExternalWritable := 'False'} : Int;   // GIN number from Fifo
      sudi_LostCounter { ExternalAccessible := 'False'; ExternalVisible := 'False'; ExternalWritable := 'False'} : UDInt;   // Counter of generated messages
      si_Location { ExternalAccessible := 'False'; ExternalVisible := 'False'; ExternalWritable := 'False'} : UInt;
   END_VAR


BEGIN
	(*
	----------------------------------------------------------------------------------------
	|                                                                                      |
	|  Copyright  2023             FORTNA Europe BV                                        |
	|  All Rights Reserved         Netherlands                                             |
	|                                                                                      |
	----------------------------------------------------------------------------------------
	Version history:
	Date        | Version   | Author       | Remark
	----------------------------------------------------------------------------------------
	30/06/2023  | 1.0       | S. Nikodem   | Release TIA 17 | DHL Munich 2023
	13/03/2024  | 1.1       | S. Nieswiec  | Added to new baseline, block needs uptade after munich is finished
	*)

	REGION 1 - Read fifo status

	    "FC_Fifo"(ic_Mode := 'S',
	              qUDT_Status => #ss_Status.FIFOStatus,
	              qx_Error => #ss_Status.FIFOError,
	              qx_Warning => #ss_Status.FIFOWarning,
	              iqv_Data := #si_GIN,
	              iqUDT_FifoHeader := #iq_UDT_FifoHeader_LostGin,
	              iqv_DataBuffer := #iqs_FifoData_LostGin);
	END_REGION

	REGION 2 - Read lost GIN

	    IF (NOT #iq_UDT_FifoHeader_LostGin.Status.Empty                             // FIFO not empty
	        AND NOT #ss_Status.FIFOError)                                          // No FIFO error
	    THEN

	        // Mode 'R' - Read FIFO record
	        "FC_Fifo"(ic_Mode := 'R',
	                  qUDT_Status => #ss_Status.FIFOStatus,
	                  qx_Error => #ss_Status.FIFOError,
	                  qx_Warning => #ss_Status.FIFOWarning,
	                  iqv_Data := #si_GIN,
	                  iqUDT_FifoHeader := #iq_UDT_FifoHeader_LostGin,
	                  iqv_DataBuffer := #iqs_FifoData_LostGin);

	        //Location
	        IF "DB_GIN".GIN[#si_GIN].DHL.ParcelLocation.Current = 0 THEN

	            #si_Location := "DB_GIN".GIN[#si_GIN].DHL.ParcelLocation.Last;
	        ELSE

	            #si_Location := "DB_GIN".GIN[#si_GIN].DHL.ParcelLocation.Current;

	        END_IF;

	        //Sort Result message - parcel lost
	        #s_FB_MFC_Sort_SortResult(is_ObjectID := "DB_GIN".GIN[#si_GIN].DHL.ObjectID,
	                                  ii_DischargeLocation := #si_Location,
	                                  ii_Result := 3,
	                                  ii_Reason := 6,
	                                  ii_SourceNode := #ii_SourceNode,
	                                  ii_DestinationNode := #ii_DestinationNode,
	                                  iq_UDT_FifoHeader := #iq_UDT_FifoHeader_MFCMessage,
	                                  iqs_FifoData := #iqs_FifoData_MFCMessage,
	                                  iqdi_MessageSequenceNumber := #iqdi_MessageSequenceNumber);


	        //Counter only for statistics
	        #sudi_LostCounter += 1;

	        //Reset
	        #si_Location := 0;
	        #si_GIN := 0;

	    END_IF;

	END_REGION
END_FUNCTION_BLOCK

FUNCTION_BLOCK "FB_Xray_BackBelt"
{ S7_Optimized_Access := 'TRUE' }
VERSION : 0.1
// ATTRIBUTES
// AUTO_NUMBER = True
// BLOCK_NUMBER = 109
// END_ATTRIBUTES
   VAR_INPUT
      i_UDT_XrayConfiguration { ExternalAccessible := 'False'; ExternalVisible := 'False'; ExternalWritable := 'False'} : "UDT_XrayRapiscanConfiguration";   // Xray configuration structure
      i_UDT_InputConveyorConfiguration { ExternalAccessible := 'False'; ExternalVisible := 'False'; ExternalWritable := 'False'} : "UDT_ConveyorConfiguration";   // Input conveyor configuration structure
      ix_Enable { ExternalAccessible := 'False'; ExternalVisible := 'False'; ExternalWritable := 'False'} : Bool;   // TRUE when function should be active
   END_VAR

   VAR_IN_OUT
      iqa_XrayConveyorTrackingData : Array[*] of Int;   // Xray conveyor tracking array
      iqa_InputConveyorTrackingData : Array[*] of Int;   // Input conveyor tracking array
      iq_UDT_XrayConveyorInterface : "UDT_ConveyorInterface";   // Xray conveyor interface structure
      iq_UDT_XrayInterface : "UDT_XrayInterface";   // Xray interface structure
   END_VAR

   VAR
      F_TRIG_ConvRunRvs {InstructionName := 'F_TRIG'; LibVersion := '1.0'; ExternalAccessible := 'False'; ExternalVisible := 'False'; ExternalWritable := 'False'; S7_SetPoint := 'False'} : F_TRIG;   // Falling edge trigger of Xray conveyor runs in reverse direction signal
      R_TRIG_BackBelt {InstructionName := 'R_TRIG'; LibVersion := '1.0'; ExternalAccessible := 'False'; ExternalVisible := 'False'; ExternalWritable := 'False'; S7_SetPoint := 'False'} : R_TRIG;   // Rising edge trigger of Backbelt signal
      sa_BackbeltDistance { ExternalAccessible := 'False'; ExternalVisible := 'False'; ExternalWritable := 'False'} : Array[1..20] of Int;   // Backbelt distances
      ss_Counter { ExternalAccessible := 'False'; ExternalVisible := 'False'; ExternalWritable := 'False'} : Struct   // Statistics counters
         InputConveyorRunRvs { ExternalAccessible := 'False'; ExternalVisible := 'False'; ExternalWritable := 'False'} : UDInt;   // Counter how many times the "InputConveyorRunRvs" signal has been activated
         XrayConveyorEnoughSpace { ExternalAccessible := 'False'; ExternalVisible := 'False'; ExternalWritable := 'False'} : UDInt;   // Counter how many times the "XrayConveyorEnoughSpace" signal has been activated
         InputConveyorNotEnoughSpace { ExternalAccessible := 'False'; ExternalVisible := 'False'; ExternalWritable := 'False'} : UDInt;   // Counter how many times the "InputConveyorNotEnoughSpace" signal has been activated
         BackbeltActive { ExternalAccessible := 'False'; ExternalVisible := 'False'; ExternalWritable := 'False'} : UDInt;   // Counter how many times the "BackbeltActive" signal has been activated
      END_STRUCT;
      si_XrayConveyorDisplacement { ExternalAccessible := 'False'; ExternalVisible := 'False'; ExternalWritable := 'False'} : Int;   // Xray conveyor displacement when conveyor running reverse
      si_ArraySavePosition { ExternalAccessible := 'False'; ExternalVisible := 'False'; ExternalWritable := 'False'} : Int := 1;   // Save position
      si_XrayConveyorGapDistance { ExternalAccessible := 'False'; ExternalVisible := 'False'; ExternalWritable := 'False'} : Int;   // Xray conveyor gap distance, from conveyor beginning to first parcel
      si_InputConveyorGapDistance { ExternalAccessible := 'False'; ExternalVisible := 'False'; ExternalWritable := 'False'} : Int;   // Input conveyor gap distance, from conveyor beginning to first parcel
      sx_InputConveyorRunRvs { ExternalAccessible := 'False'; ExternalVisible := 'False'; ExternalWritable := 'False'} : Bool;   // Request command to run reverse input conveyor
   END_VAR

   VAR_TEMP
      ti_XrayConveyor : Int;   // Loop counter - to check gap between parcel and beginning of the Xray conveyor
      ti_InputConveyor : Int;   // Loop counter - to check gap between parcel and beginning of the input conveyor
      ti_ArrayElements : Int;   // Copy size of the array
   END_VAR


BEGIN
	(*
	----------------------------------------------------------------------------------------
	|                                                                                      |
	|  Copyright  2023             FORTNA Europe BV                                        |
	|  All Rights Reserved         Netherlands                                             |
	|                                                                                      |
	----------------------------------------------------------------------------------------

	Version history:
	Date        | Version   | Author       | Remark
	----------------------------------------------------------------------------------------
	07/03/2023  | 1.0       | S. Nikodem   | Release TIA 17 | DHL Munich 2023
	13/03/2024  | 1.1       | S. Nieswiec  | Added to new baseline
	02/05/2024  | 1.2       | J.Majer      | Datatype conversions changed from automatic to explicit, to accomodate IEC 61131-3 standard
	*)

	REGION 1 - Triggers

	    // Xray conveyor running in reverse direction
	    #F_TRIG_ConvRunRvs(CLK := #iq_UDT_XrayInterface.XrayConveyor.RunRvs);

	    // BackBelt active
	    #R_TRIG_BackBelt(CLK := #iq_UDT_XrayInterface.Backbelt.Active);

	    IF #R_TRIG_BackBelt.Q THEN

	        //Only for statistics
	        #ss_Counter.BackbeltActive += 1;

	    END_IF;

	END_REGION

	REGION 2 - Function enable

	    //Copy signal to Xray interface
	    #iq_UDT_XrayInterface.Backbelt.Enable := #ix_Enable;

	END_REGION

	REGION 3 - Check if is enough space for Backbelt

	    IF #R_TRIG_BackBelt.Q                                  //Rising edge trigger active
	        AND #ix_Enable                                      //Function is enable
	    THEN

	        //Initial variable
	        #si_XrayConveyorGapDistance := 0;
	        #si_InputConveyorGapDistance := 0;

	        //Check the gap between parcel and beginning of the Xray conveyor
	        FOR #ti_XrayConveyor := DINT_TO_INT(#i_UDT_XrayConfiguration.XrayConveyor.Length) TO 0 BY -1
	        DO

	            #si_XrayConveyorGapDistance += 1;


	            IF #iqa_XrayConveyorTrackingData[#ti_XrayConveyor] > 0 THEN

	                //Parcel detected, exit the loop
	                EXIT;

	            END_IF;

	        END_FOR;

	        //Check if there is
	        IF #si_XrayConveyorGapDistance < #i_UDT_XrayConfiguration.BackBeltDistance THEN

	            //Check the gap between parcel and beginning of the Input conveyor
	            FOR #ti_InputConveyor := DINT_TO_INT(#i_UDT_InputConveyorConfiguration.Common.Length) TO 0 BY -1
	            DO

	                #si_InputConveyorGapDistance += 1;

	                IF #iqa_InputConveyorTrackingData[#ti_InputConveyor] > 0 THEN

	                    //Parcel detected, exit the loop
	                    EXIT;

	                END_IF;

	            END_FOR;


	            IF #si_InputConveyorGapDistance > #i_UDT_XrayConfiguration.BackBeltDistance THEN

	                //Run input conveyor in reverse direction if needed
	                #sx_InputConveyorRunRvs := True;

	                //Only for statistics
	                #ss_Counter.InputConveyorRunRvs += 1;

	            ELSE

	                //Only for statistics
	                #ss_Counter.InputConveyorNotEnoughSpace += 1;

	            END_IF;

	        ELSE

	            //Only for statistics
	            #ss_Counter.XrayConveyorEnoughSpace += 1;

	        END_IF;

	    END_IF;

	END_REGION

	REGION 4 - Input conveyor control

	    //Control command to run input conveyor in reverse direction
	    #iq_UDT_XrayInterface.InputConveyor.CommandRunRvs := #sx_InputConveyorRunRvs
	    AND #iq_UDT_XrayInterface.XrayConveyor.RunRvs
	    AND #iq_UDT_XrayInterface.Backbelt.Active
	    AND #ix_Enable;

	    //Reset command
	    IF NOT #ix_Enable
	        OR NOT #iq_UDT_XrayInterface.Backbelt.Active
	    THEN
	        #sx_InputConveyorRunRvs := False;
	    END_IF;

	END_REGION

	REGION 5 - Save Backbelt distance

	    //Logic prepared only for commissioning

	    //Count up value from displacement to static variable
	    IF #iq_UDT_XrayInterface.XrayConveyor.RunRvs THEN
	        #si_XrayConveyorDisplacement += ABS(#iq_UDT_XrayConveyorInterface.Displacement);
	    END_IF;

	    //When reverse direction is switch off then copy data to array
	    IF #F_TRIG_ConvRunRvs.Q THEN
	        //Copy value to array
	        #sa_BackbeltDistance[#si_ArraySavePosition] := #si_XrayConveyorDisplacement;

	        //Switch up save position in array
	        #si_ArraySavePosition += 1;

	        //Reset value in variable
	        #si_XrayConveyorDisplacement := 0;
	    END_IF;

	    // Get size of the array.
	    #ti_ArrayElements := "FC_GetNrOfArrayEl"(#sa_BackbeltDistance);

	    //Reset saving position
	    IF #ti_ArrayElements > #si_ArraySavePosition THEN

	        #si_ArraySavePosition := 1;

	    END_IF;

	END_REGION
END_FUNCTION_BLOCK

FUNCTION_BLOCK "FB_Xray_RegistrationInfo"
{ S7_Optimized_Access := 'TRUE' }
VERSION : 0.1
// ATTRIBUTES
// AUTO_NUMBER = True
// BLOCK_NUMBER = 111
// END_ATTRIBUTES
   VAR_INPUT
      ii_GINRangeStart { ExternalAccessible := 'False'; ExternalVisible := 'False'; ExternalWritable := 'False'} : Int;   // GIN range start value
      ii_GINRangeEnd { ExternalAccessible := 'False'; ExternalVisible := 'False'; ExternalWritable := 'False'} : Int;   // GIN range end value
   END_VAR

   VAR_IN_OUT
      iqs_XrayRegistrationInfo : Struct   // Structure from MFC
         ObjectID : String[10];   // ObjectI D
         VID : String[16];   // VID
         PieceID : String[40];   // Piece ID
         RoutingCode : String[2];   // Routing code
      END_STRUCT;
   END_VAR

   VAR
      ss_Counter { ExternalAccessible := 'False'; ExternalVisible := 'False'; ExternalWritable := 'False'} : Struct   // Counterts only for statistics
         SavedData { ExternalAccessible := 'False'; ExternalVisible := 'False'; ExternalWritable := 'False'} : ULInt;   // Counter of saved data
         DataNotMerged { ExternalAccessible := 'False'; ExternalVisible := 'False'; ExternalWritable := 'False'} : ULInt;   // Counter of triggers when  data not merged
      END_STRUCT;
      ss_OldObjectID { ExternalAccessible := 'False'; ExternalVisible := 'False'; ExternalWritable := 'False'} : String[10];   // Old Objcet ID
      sx_NewData { ExternalAccessible := 'False'; ExternalVisible := 'False'; ExternalWritable := 'False'} : Bool;   // New Object ID
      sx_DataMerged { ExternalAccessible := 'False'; ExternalVisible := 'False'; ExternalWritable := 'False'} : Bool;   // Data merged
   END_VAR

   VAR_TEMP
      ti_Loop_GIN : Int;
   END_VAR


BEGIN
	(*
	----------------------------------------------------------------------------------------
	|                                                                                      |
	|  Copyright  2023             FORTNA Europe BV                                        |
	|  All Rights Reserved         Netherlands                                             |
	|                                                                                      |
	----------------------------------------------------------------------------------------
	Version history:
	Date        | Version   | Author       | Remark
	----------------------------------------------------------------------------------------
	28/04/2023  | 1.0       | S. Nikodem   | Release TIA 17 | DHL Munich 2023
	13/03/2024  | 1.1       | S. Nieswiec  | Added to new baseline
	*)

	REGION 1 - New data

	    IF #iqs_XrayRegistrationInfo.ObjectID <> #ss_OldObjectID THEN

	        //Set variable
	        #sx_NewData := TRUE;
	        //Copy value to memory
	        #ss_OldObjectID := #iqs_XrayRegistrationInfo.ObjectID;

	    END_IF;

	END_REGION

	REGION 2 - Save value in array row

	    IF #sx_NewData THEN

	        FOR #ti_Loop_GIN := #ii_GINRangeStart TO #ii_GINRangeEnd DO

	            IF "DB_GIN".GIN[#ti_Loop_GIN].DHL.ObjectID = #iqs_XrayRegistrationInfo.ObjectID THEN

	                //VID
	                "DB_GIN".GIN[#ti_Loop_GIN].DHL.VID := #iqs_XrayRegistrationInfo.VID;
	                //PieceID
	                "DB_GIN".GIN[#ti_Loop_GIN].DHL.PieceID := #iqs_XrayRegistrationInfo.PieceID;
	                //RoutingCode
	                "DB_GIN".GIN[#ti_Loop_GIN].DHL.Xray.RoutingCode := #iqs_XrayRegistrationInfo.RoutingCode;

	                //Counterts only for statistics
	                #ss_Counter.SavedData += 1;

	                //Data merged
	                #sx_DataMerged := TRUE;

	                //Exit loop
	                EXIT;

	            END_IF;

	        END_FOR;

	        IF NOT #sx_DataMerged THEN

	            //Counterts only for statistics
	            #ss_Counter.DataNotMerged += 1;

	        END_IF;

	        //Reset value
	        #sx_NewData := FALSE;
	        #sx_DataMerged := FALSE;

	    END_IF;

	END_REGION

END_FUNCTION_BLOCK

FUNCTION_BLOCK "FB_Xray_SerialCommunication"
{ S7_Optimized_Access := 'TRUE' }
VERSION : 0.1
// ATTRIBUTES
// AUTO_NUMBER = True
// BLOCK_NUMBER = 112
// END_ATTRIBUTES
   VAR_INPUT
      i_UDT_SerialCommunicationConfiguration { ExternalAccessible := 'False'; ExternalVisible := 'False'; ExternalWritable := 'False'} : "UDT_SerialComConfiguration";   // Serial communication configuration
      ix_Trigger { ExternalAccessible := 'False'; ExternalVisible := 'False'; ExternalWritable := 'False'} : Bool;   // Diagnostics trigger signal - Connect system memory clock
   END_VAR

   VAR_OUTPUT
      q_UDT_Status { ExternalAccessible := 'False'; ExternalVisible := 'False'; ExternalWritable := 'False'} : "UDT_SerialCommunicationStatus";   // Status structure
   END_VAR

   VAR_IN_OUT
      iq_UDT_XrayInterface : "UDT_XrayInterface";   // Xray interface structure
   END_VAR

   VAR
      Signal_Get {InstructionName := 'Signal_Get'; LibVersion := '4.0'; ExternalAccessible := 'False'; ExternalVisible := 'False'; ExternalWritable := 'False'; S7_SetPoint := 'False'} : Signal_Get;   // Signal_get block
      ss_Status { ExternalAccessible := 'False'; ExternalVisible := 'False'; ExternalWritable := 'False'} : Struct   // Status structure
         NDR { ExternalAccessible := 'False'; ExternalVisible := 'False'; ExternalWritable := 'False'} : Bool;
         Error { ExternalAccessible := 'False'; ExternalVisible := 'False'; ExternalWritable := 'False'} : Bool;
         Status { ExternalAccessible := 'False'; ExternalVisible := 'False'; ExternalWritable := 'False'} : Word;
         DTR { ExternalAccessible := 'False'; ExternalVisible := 'False'; ExternalWritable := 'False'} : Bool;
         DSR { ExternalAccessible := 'False'; ExternalVisible := 'False'; ExternalWritable := 'False'} : Bool;
         RTS { ExternalAccessible := 'False'; ExternalVisible := 'False'; ExternalWritable := 'False'} : Bool;
         CTS { ExternalAccessible := 'False'; ExternalVisible := 'False'; ExternalWritable := 'False'} : Bool;
         DCD { ExternalAccessible := 'False'; ExternalVisible := 'False'; ExternalWritable := 'False'} : Bool;
         RING { ExternalAccessible := 'False'; ExternalVisible := 'False'; ExternalWritable := 'False'} : Bool;
      END_STRUCT;
   END_VAR


BEGIN
	(*
	----------------------------------------------------------------------------------------
	|                                                                                      |
	|  Copyright  2023             FORTNA Europe BV                                        |
	|  All Rights Reserved         Netherlands                                             |
	|                                                                                      |
	----------------------------------------------------------------------------------------
	Version history:
	Date        | Version   | Author       | Remark
	----------------------------------------------------------------------------------------
	16/03/2023  | 1.0       | S. Nikodem   | Release TIA 17 | DHL Munich 2023
	13/03/2024  | 1.1       | S. Nieswiec  | Added to new baseline
	*)

	REGION 1 - P2P diagnostics function

	    #Signal_Get(REQ := #ix_Trigger,
	                "PORT" := #i_UDT_SerialCommunicationConfiguration."Port",
	                NDR => #ss_Status.NDR,
	                ERROR => #ss_Status.Error,
	                STATUS => #ss_Status.Status,
	                DTR => #ss_Status.DTR,
	                DSR => #ss_Status.DSR,
	                RTS => #ss_Status.RTS,
	                CTS => #ss_Status.CTS,
	                DCD => #ss_Status.DCD,
	                RING => #ss_Status.RING);

	END_REGION

	REGION 2 - Status structure

	    //Output structure
	    #q_UDT_Status.Connected := #ss_Status.DSR AND #ss_Status.CTS;

	    #q_UDT_Status.CommunicationFault := #ss_Status.Error
	    OR NOT #ss_Status.DSR
	    OR NOT #ss_Status.CTS;

	    //In/Out structure
	    #iq_UDT_XrayInterface.Communication.Connceted := #ss_Status.DSR AND #ss_Status.CTS;

	END_REGION

END_FUNCTION_BLOCK

FUNCTION_BLOCK "FB_XbeltExit_Interface"
{ S7_Optimized_Access := 'TRUE' }
VERSION : 2.0
// ATTRIBUTES
// AUTO_NUMBER = True
// BLOCK_NUMBER = 108
// END_ATTRIBUTES
   VAR_INPUT
      i_UDT_Sorter_Downstream { ExternalAccessible := 'False'; ExternalVisible := 'False'; ExternalWritable := 'False'} : "Sorter_DownStream_Advanced";   // Downstream Sorter input
      i_UDT_Outfeed2StatesStatus { ExternalAccessible := 'False'; ExternalVisible := 'False'; ExternalWritable := 'False'} : "UDT_Outfeed2StatesStatus";   // Outfeed2States
      i_UDT_AssociatedConveyorInterface { ExternalAccessible := 'False'; ExternalVisible := 'False'; ExternalWritable := 'False'} : "UDT_ConveyorInterface";   // Conveyor Interface
      ix_ConfigHorizontalOutfeed { ExternalAccessible := 'False'; ExternalVisible := 'False'; ExternalWritable := 'False'} : Bool;   // TRUE when this block is used for horizontal outfeed , FALSE for spiral
      ix_HorOutfeed_PECBoS { ExternalAccessible := 'False'; ExternalVisible := 'False'; ExternalWritable := 'False'} : Bool;   // sensor PEC begin of section
      ix_HorOutfeed_PECJam { ExternalAccessible := 'False'; ExternalVisible := 'False'; ExternalWritable := 'False'} : Bool;   // sensor PEC jam
   END_VAR

   VAR_OUTPUT
      q_UDT_Downstream_Sorter { ExternalAccessible := 'False'; ExternalVisible := 'False'; ExternalWritable := 'False'} : "DownStream_Sorter_Basic";   // Downstream Sorter output
      q_UDT_XBeltExitStatus { ExternalAccessible := 'False'; ExternalVisible := 'False'; ExternalWritable := 'False'} : "UDT_XBeltExitStatus";   // XBelt exit status
      q_UDT_XBeltExitInterface { ExternalAccessible := 'False'; ExternalVisible := 'False'; ExternalWritable := 'False'} : "UDT_XbeltExitInterface";   // XBelt exit interface
   END_VAR

   VAR_IN_OUT
      iq_UDT_ChuteExternalHandshake : "UDT_ConveyorHandshake";   // Chute handshake
   END_VAR

   VAR
      s_UDT_Downstream_Sorter { ExternalAccessible := 'False'; ExternalVisible := 'False'; ExternalWritable := 'False'; S7_SetPoint := 'False'} : "DownStream_Sorter_Basic";   // static Downstream Sorter status
      s_UDT_XBeltExitStatus { ExternalAccessible := 'False'; ExternalVisible := 'False'; ExternalWritable := 'False'; S7_SetPoint := 'False'} : "UDT_XBeltExitStatus";   // static X-Belt exit status
      s_UDT_XBeltExitInterface { ExternalAccessible := 'False'; ExternalVisible := 'False'; ExternalWritable := 'False'; S7_SetPoint := 'False'} : "UDT_XbeltExitInterface";   // static X-Belt exit interface
      sa_ExchangeObjectID { ExternalAccessible := 'False'; ExternalVisible := 'False'; ExternalWritable := 'False'} : Array[0..1] of DInt;   // static exchange object ID
   END_VAR

   VAR CONSTANT
      c_MaximumLength : DInt := 5000;   // Maximum lenght
   END_VAR


BEGIN
	(*
	----------------------------------------------------------------------------------------
	|                                                                                      |
	|  Copyright  2023             FORTNA Europe BV                                        |
	|  All Rights Reserved         Netherlands                                             |
	|                                                                                      |
	----------------------------------------------------------------------------------------

